Yaskawa INFORM job: DEMO_ROOF_UPPER_0625_3PAINT_22.JBI

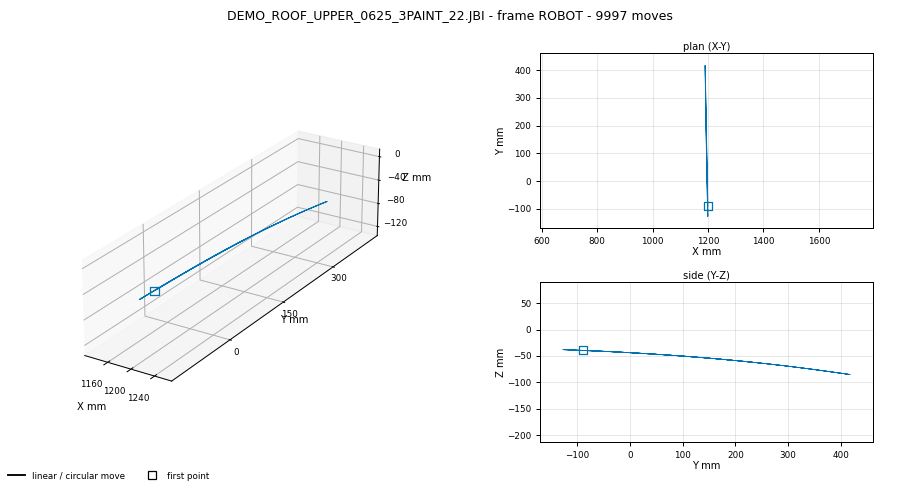
[picture p0: tool path of DEMO_ROOF_UPPER_0625_3PAINT_22.JBI in frame ROBOT, 9997 of 9997 moves have a stored position in this frame; points joined in program order, loops and branches not executed]
/JOB
//NAME DEMO_ROOF_UPPER_0625_3PAINT22
//POS
///NPOS 9997,0,0,0,0,0
///TOOL 0
///USER 0
///POSTYPE ROBOT
///RECTAN
///RCONF 1,0,0,0,0,0,0,0,0,0,0,0,0,0,0,0,0,0,0,0,0,0,0,0
C00000=1199.576,-89.571,-39.322,179.341,5.541,149.171
C00001=1199.572,-89.321,-39.332,179.344,5.541,149.171
C00002=1199.567,-89.072,-39.342,179.346,5.541,149.170
C00003=1199.562,-88.822,-39.354,179.348,5.541,149.169
C00004=1199.556,-88.573,-39.364,179.350,5.541,149.169
C00005=1199.551,-88.322,-39.375,179.353,5.541,149.168
C00006=1199.546,-88.073,-39.385,179.355,5.541,149.167
C00007=1199.540,-87.823,-39.395,179.357,5.542,149.167
C00008=1199.535,-87.573,-39.406,179.359,5.542,149.166
C00009=1199.530,-87.324,-39.416,179.362,5.542,149.165
C00010=1199.525,-87.074,-39.427,179.365,5.542,149.165
C00011=1199.519,-86.824,-39.437,179.366,5.542,149.164
C00012=1199.514,-86.574,-39.448,179.369,5.543,149.163
C00013=1199.509,-86.325,-39.458,179.371,5.542,149.163
C00014=1199.504,-86.075,-39.469,179.374,5.543,149.162
C00015=1199.498,-85.825,-39.480,179.375,5.543,149.162
C00016=1199.493,-85.575,-39.490,179.378,5.543,149.161
C00017=1199.488,-85.326,-39.500,179.381,5.544,149.160
C00018=1199.483,-85.076,-39.512,179.383,5.543,149.159
C00019=1199.477,-84.826,-39.522,179.385,5.544,149.159
C00020=1199.472,-84.576,-39.532,179.387,5.544,149.158
C00021=1199.467,-84.327,-39.543,179.390,5.544,149.158
C00022=1199.462,-84.077,-39.554,179.392,5.544,149.157
C00023=1199.457,-83.827,-39.564,179.394,5.545,149.156
C00024=1199.452,-83.577,-39.575,179.397,5.545,149.156
C00025=1199.446,-83.328,-39.586,179.399,5.545,149.155
C00026=1199.441,-83.078,-39.596,179.401,5.545,149.154
C00027=1199.436,-82.828,-39.606,179.403,5.545,149.154
C00028=1199.431,-82.579,-39.618,179.406,5.545,149.153
C00029=1199.425,-82.329,-39.628,179.408,5.545,149.152
C00030=1199.420,-82.079,-39.638,179.410,5.546,149.152
C00031=1199.415,-81.830,-39.649,179.412,5.546,149.151
C00032=1199.410,-81.580,-39.660,179.415,5.546,149.150
C00033=1199.404,-81.330,-39.670,179.417,5.546,149.150
C00034=1199.400,-81.081,-39.681,179.419,5.546,149.149
C00035=1199.394,-80.831,-39.692,179.422,5.547,149.149
C00036=1199.388,-80.581,-39.703,179.424,5.546,149.148
C00037=1199.383,-80.332,-39.714,179.426,5.547,149.147
C00038=1199.378,-80.081,-39.724,179.429,5.547,149.146
C00039=1199.373,-79.833,-39.735,179.431,5.547,149.146
C00040=1199.368,-79.582,-39.746,179.433,5.548,149.145
C00041=1199.362,-79.333,-39.756,179.435,5.547,149.145
C00042=1199.358,-79.083,-39.767,179.438,5.548,149.144
C00043=1199.353,-78.833,-39.778,179.440,5.548,149.143
C00044=1199.347,-78.584,-39.789,179.442,5.548,149.143
C00045=1199.342,-78.333,-39.800,179.445,5.549,149.142
C00046=1199.336,-78.084,-39.811,179.447,5.548,149.141
C00047=1199.331,-77.834,-39.821,179.450,5.549,149.140
C00048=1199.326,-77.585,-39.832,179.451,5.549,149.140
C00049=1199.321,-77.335,-39.843,179.454,5.549,149.139
C00050=1199.316,-77.085,-39.854,179.457,5.550,149.139
C00051=1199.310,-76.836,-39.865,179.459,5.549,149.138
C00052=1199.305,-76.585,-39.876,179.461,5.550,149.137
C00053=1199.300,-76.336,-39.887,179.463,5.550,149.137
C00054=1199.295,-76.086,-39.897,179.466,5.550,149.136
C00055=1199.289,-75.837,-39.908,179.468,5.550,149.135
C00056=1199.284,-75.566,-39.920,179.470,5.550,149.135
C00057=1199.278,-75.295,-39.933,179.473,5.551,149.134
C00058=1199.272,-75.024,-39.944,179.476,5.551,149.133
C00059=1199.267,-74.754,-39.955,179.478,5.551,149.132
C00060=1199.262,-74.504,-39.967,179.480,5.551,149.132
C00061=1199.256,-74.254,-39.977,179.483,5.552,149.131
C00062=1199.251,-74.005,-39.989,179.485,5.551,149.131
C00063=1199.246,-73.754,-39.999,179.487,5.552,149.130
C00064=1199.241,-73.505,-40.010,179.489,5.552,149.129
C00065=1199.235,-73.255,-40.022,179.492,5.552,149.129
C00066=1199.230,-73.006,-40.032,179.494,5.553,149.128
C00067=1199.225,-72.756,-40.044,179.496,5.552,149.127
C00068=1199.220,-72.506,-40.054,179.499,5.553,149.127
C00069=1199.214,-72.257,-40.066,179.501,5.554,149.126
C00070=1199.209,-72.007,-40.077,179.503,5.553,149.125
C00071=1199.204,-71.757,-40.088,179.506,5.554,149.125
C00072=1199.198,-71.508,-40.099,179.508,5.553,149.124
C00073=1199.194,-71.258,-40.110,179.511,5.554,149.123
C00074=1199.189,-71.008,-40.121,179.513,5.555,149.123
C00075=1199.183,-70.759,-40.132,179.515,5.554,149.122
C00076=1199.178,-70.508,-40.143,179.518,5.555,149.121
C00077=1199.173,-70.259,-40.154,179.520,5.554,149.121
C00078=1199.168,-70.010,-40.165,179.522,5.555,149.120
C00079=1199.162,-69.759,-40.176,179.525,5.556,149.119
C00080=1199.157,-69.510,-40.188,179.527,5.555,149.119
C00081=1199.152,-69.261,-40.199,179.529,5.556,149.118
C00082=1199.146,-69.011,-40.211,179.532,5.555,149.117
C00083=1199.141,-68.761,-40.221,179.534,5.556,149.117
C00084=1199.136,-68.512,-40.232,179.536,5.556,149.116
C00085=1199.131,-68.262,-40.244,179.538,5.556,149.115
C00086=1199.126,-68.011,-40.255,179.541,5.557,149.115
C00087=1199.121,-67.762,-40.266,179.544,5.557,149.114
C00088=1199.115,-67.513,-40.277,179.545,5.557,149.114
C00089=1199.110,-67.263,-40.289,179.548,5.557,149.113
C00090=1199.105,-67.013,-40.299,179.550,5.557,149.112
C00091=1199.099,-66.763,-40.311,179.553,5.557,149.111
C00092=1199.095,-66.514,-40.322,179.555,5.558,149.111
C00093=1199.089,-66.264,-40.334,179.557,5.558,149.110
C00094=1199.084,-66.014,-40.345,179.560,5.558,149.110
C00095=1199.079,-65.765,-40.355,179.562,5.559,149.109
C00096=1199.073,-65.515,-40.367,179.564,5.558,149.108
C00097=1199.069,-65.265,-40.379,179.567,5.559,149.108
C00098=1199.063,-65.015,-40.390,179.569,5.559,149.107
C00099=1199.058,-64.766,-40.401,179.571,5.559,149.106
C00100=1199.053,-64.516,-40.412,179.574,5.560,149.105
C00101=1199.048,-64.266,-40.424,179.576,5.559,149.105
C00102=1199.043,-64.017,-40.435,179.578,5.560,149.104
C00103=1199.037,-63.767,-40.447,179.581,5.561,149.104
C00104=1199.032,-63.518,-40.458,179.583,5.560,149.103
C00105=1199.027,-63.268,-40.470,179.586,5.561,149.102
C00106=1199.022,-63.018,-40.481,179.588,5.560,149.101
C00107=1199.016,-62.769,-40.491,179.590,5.561,149.101
C00108=1199.011,-62.519,-40.503,179.593,5.562,149.100
C00109=1199.006,-62.269,-40.515,179.595,5.561,149.100
C00110=1199.001,-62.019,-40.526,179.597,5.562,149.099
C00111=1198.996,-61.769,-40.538,179.600,5.562,149.098
C00112=1198.990,-61.520,-40.549,179.602,5.562,149.098
C00113=1198.985,-61.271,-40.560,179.604,5.563,149.097
C00114=1198.980,-61.021,-40.572,179.607,5.563,149.096
C00115=1198.975,-60.771,-40.584,179.609,5.563,149.096
C00116=1198.970,-60.521,-40.596,179.612,5.563,149.095
C00117=1198.965,-60.272,-40.606,179.614,5.564,149.094
C00118=1198.959,-60.022,-40.618,179.616,5.564,149.094
C00119=1198.955,-59.773,-40.630,179.619,5.564,149.093
C00120=1198.949,-59.523,-40.642,179.621,5.564,149.092
C00121=1198.944,-59.272,-40.652,179.623,5.564,149.092
C00122=1198.939,-59.022,-40.664,179.626,5.565,149.091
C00123=1198.933,-58.774,-40.675,179.628,5.565,149.090
C00124=1198.928,-58.524,-40.687,179.630,5.565,149.090
C00125=1198.923,-58.274,-40.698,179.633,5.565,149.089
C00126=1198.918,-58.025,-40.711,179.635,5.565,149.088
C00127=1198.913,-57.775,-40.723,179.637,5.566,149.088
C00128=1198.908,-57.525,-40.734,179.640,5.566,149.087
C00129=1198.902,-57.276,-40.745,179.642,5.566,149.086
C00130=1198.897,-57.026,-40.757,179.645,5.566,149.086
C00131=1198.892,-56.776,-40.769,179.647,5.567,149.085
C00132=1198.887,-56.527,-40.780,179.649,5.567,149.085
C00133=1198.882,-56.277,-40.792,179.652,5.567,149.084
C00134=1198.876,-56.027,-40.804,179.654,5.568,149.083
C00135=1198.872,-55.777,-40.815,179.656,5.567,149.082
C00136=1198.866,-55.527,-40.827,179.659,5.568,149.082
C00137=1198.861,-55.278,-40.838,179.661,5.569,149.081
C00138=1198.855,-55.028,-40.850,179.663,5.568,149.081
C00139=1198.850,-54.778,-40.861,179.666,5.569,149.080
C00140=1198.846,-54.529,-40.873,179.669,5.569,149.079
C00141=1198.840,-54.280,-40.885,179.671,5.569,149.078
C00142=1198.836,-54.030,-40.897,179.673,5.569,149.078
C00143=1198.830,-53.780,-40.909,179.676,5.570,149.077
C00144=1198.825,-53.530,-40.920,179.678,5.570,149.077
C00145=1198.820,-53.280,-40.932,179.680,5.570,149.076
C00146=1198.815,-53.030,-40.944,179.683,5.571,149.075
C00147=1198.809,-52.781,-40.956,179.685,5.570,149.074
C00148=1198.805,-52.531,-40.968,179.687,5.571,149.074
C00149=1198.799,-52.282,-40.979,179.690,5.572,149.073
C00150=1198.793,-52.032,-40.991,179.692,5.571,149.073
C00151=1198.789,-51.783,-41.002,179.695,5.572,149.072
C00152=1198.783,-51.533,-41.015,179.697,5.572,149.071
C00153=1198.778,-51.283,-41.027,179.699,5.572,149.071
C00154=1198.773,-51.034,-41.038,179.702,5.573,149.070
C00155=1198.768,-50.784,-41.050,179.704,5.573,149.069
C00156=1198.762,-50.534,-41.062,179.706,5.573,149.069
C00157=1198.757,-50.285,-41.074,179.709,5.573,149.068
C00158=1198.753,-50.035,-41.086,179.711,5.574,149.067
C00159=1198.747,-49.785,-41.098,179.713,5.574,149.067
C00160=1198.742,-49.515,-41.110,179.716,5.574,149.066
C00161=1198.736,-49.245,-41.123,179.719,5.575,149.065
C00162=1198.731,-48.975,-41.136,179.721,5.575,149.065
C00163=1198.725,-48.705,-41.149,179.724,5.575,149.064
C00164=1198.720,-48.456,-41.161,179.726,5.575,149.063
C00165=1198.714,-48.206,-41.173,179.729,5.576,149.062
C00166=1198.709,-47.956,-41.185,179.731,5.576,149.062
C00167=1198.704,-47.706,-41.196,179.733,5.576,149.061
C00168=1198.699,-47.457,-41.209,179.736,5.576,149.060
C00169=1198.694,-47.207,-41.221,179.738,5.577,149.060
C00170=1198.688,-46.957,-41.233,179.741,5.577,149.059
C00171=1198.683,-46.708,-41.245,179.743,5.577,149.058
C00172=1198.678,-46.458,-41.257,179.746,5.577,149.058
C00173=1198.673,-46.209,-41.269,179.748,5.578,149.057
C00174=1198.668,-45.959,-41.281,179.750,5.578,149.057
C00175=1198.662,-45.709,-41.293,179.753,5.578,149.056
C00176=1198.657,-45.460,-41.306,179.755,5.579,149.055
C00177=1198.653,-45.210,-41.317,179.757,5.578,149.054
C00178=1198.647,-44.960,-41.329,179.760,5.579,149.054
C00179=1198.642,-44.711,-41.341,179.763,5.579,149.053
C00180=1198.637,-44.461,-41.353,179.764,5.579,149.053
C00181=1198.632,-44.211,-41.366,179.767,5.580,149.052
C00182=1198.627,-43.961,-41.378,179.770,5.580,149.051
C00183=1198.622,-43.712,-41.390,179.772,5.581,149.051
C00184=1198.617,-43.462,-41.402,179.774,5.580,149.050
C00185=1198.611,-43.212,-41.414,179.777,5.581,149.049
C00186=1198.606,-42.963,-41.426,179.779,5.582,149.049
C00187=1198.601,-42.713,-41.438,179.781,5.581,149.048
C00188=1198.596,-42.463,-41.451,179.784,5.582,149.047
C00189=1198.590,-42.213,-41.463,179.787,5.582,149.047
C00190=1198.585,-41.964,-41.475,179.789,5.583,149.046
C00191=1198.580,-41.714,-41.487,179.791,5.583,149.045
C00192=1198.575,-41.465,-41.499,179.794,5.583,149.045
C00193=1198.570,-41.215,-41.511,179.796,5.584,149.044
C00194=1198.565,-40.966,-41.524,179.798,5.583,149.043
C00195=1198.559,-40.716,-41.536,179.801,5.584,149.043
C00196=1198.555,-40.466,-41.549,179.804,5.584,149.042
C00197=1198.549,-40.216,-41.561,179.806,5.585,149.041
C00198=1198.544,-39.967,-41.573,179.808,5.585,149.041
C00199=1198.539,-39.717,-41.586,179.811,5.585,149.040
C00200=1198.534,-39.467,-41.598,179.813,5.586,149.039
C00201=1198.529,-39.218,-41.610,179.815,5.585,149.039
C00202=1198.523,-38.968,-41.622,179.817,5.586,149.038
C00203=1198.518,-38.719,-41.635,179.820,5.587,149.037
C00204=1198.513,-38.469,-41.647,179.823,5.587,149.037
C00205=1198.507,-38.220,-41.659,179.825,5.587,149.036
C00206=1198.503,-37.970,-41.672,179.828,5.587,149.035
C00207=1198.497,-37.720,-41.684,179.830,5.588,149.035
C00208=1198.492,-37.470,-41.697,179.832,5.588,149.034
C00209=1198.487,-37.221,-41.709,179.834,5.588,149.033
C00210=1198.482,-36.971,-41.721,179.837,5.589,149.033
C00211=1198.477,-36.722,-41.734,179.840,5.589,149.032
C00212=1198.471,-36.472,-41.746,179.842,5.589,149.031
C00213=1198.467,-36.222,-41.759,179.845,5.589,149.031
C00214=1198.462,-35.973,-41.771,179.847,5.590,149.030
C00215=1198.456,-35.723,-41.783,179.849,5.590,149.029
C00216=1198.451,-35.473,-41.796,179.851,5.590,149.029
C00217=1198.446,-35.224,-41.808,179.854,5.591,149.028
C00218=1198.441,-34.975,-41.821,179.857,5.591,149.027
C00219=1198.436,-34.724,-41.833,179.859,5.592,149.027
C00220=1198.431,-34.475,-41.846,179.861,5.592,149.026
C00221=1198.426,-34.225,-41.858,179.864,5.592,149.026
C00222=1198.420,-33.975,-41.870,179.866,5.592,149.025
C00223=1198.415,-33.726,-41.883,179.869,5.593,149.024
C00224=1198.410,-33.477,-41.895,179.871,5.593,149.023
C00225=1198.406,-33.227,-41.908,179.873,5.593,149.023
C00226=1198.400,-32.977,-41.920,179.876,5.594,149.022
C00227=1198.395,-32.728,-41.933,179.879,5.594,149.022
C00228=1198.389,-32.478,-41.946,179.881,5.594,149.021
C00229=1198.384,-32.229,-41.959,179.883,5.594,149.020
C00230=1198.379,-31.978,-41.971,179.886,5.595,149.019
C00231=1198.374,-31.729,-41.984,179.888,5.596,149.019
C00232=1198.369,-31.479,-41.996,179.890,5.595,149.018
C00233=1198.364,-31.230,-42.009,179.893,5.596,149.018
C00234=1198.359,-30.980,-42.022,179.896,5.596,149.017
C00235=1198.354,-30.731,-42.034,179.898,5.597,149.016
C00236=1198.349,-30.481,-42.046,179.900,5.597,149.016
C00237=1198.343,-30.231,-42.059,179.902,5.597,149.015
C00238=1198.338,-29.982,-42.072,179.905,5.598,149.014
C00239=1198.333,-29.732,-42.085,179.908,5.598,149.014
C00240=1198.328,-29.482,-42.098,179.910,5.598,149.013
C00241=1198.323,-29.233,-42.110,179.913,5.598,149.012
C00242=1198.318,-28.984,-42.123,179.915,5.599,149.012
C00243=1198.312,-28.733,-42.136,179.917,5.600,149.011
C00244=1198.307,-28.484,-42.148,179.919,5.599,149.010
C00245=1198.302,-28.234,-42.161,179.922,5.600,149.010
C00246=1198.298,-27.984,-42.174,179.925,5.600,149.009
C00247=1198.292,-27.735,-42.186,179.927,5.601,149.008
C00248=1198.287,-27.485,-42.200,179.929,5.601,149.008
C00249=1198.281,-27.236,-42.212,179.932,5.601,149.007
C00250=1198.277,-26.986,-42.225,179.934,5.602,149.006
C00251=1198.272,-26.737,-42.238,179.937,5.602,149.006
C00252=1198.267,-26.487,-42.250,179.940,5.603,149.005
C00253=1198.261,-26.237,-42.264,179.942,5.602,149.004
C00254=1198.256,-25.988,-42.276,179.944,5.603,149.004
C00255=1198.251,-25.738,-42.289,179.947,5.604,149.003
C00256=1198.246,-25.489,-42.302,179.949,5.604,149.002
C00257=1198.241,-25.239,-42.315,179.951,5.604,149.002
C00258=1198.236,-24.989,-42.328,179.954,5.604,149.001
C00259=1198.230,-24.740,-42.340,179.956,5.605,149.001
C00260=1198.226,-24.490,-42.353,179.959,5.606,149.000
C00261=1198.220,-24.240,-42.367,179.961,5.606,148.999
C00262=1198.215,-23.991,-42.379,179.964,5.606,148.999
C00263=1198.210,-23.741,-42.392,179.966,5.606,148.998
C00264=1198.204,-23.472,-42.406,179.969,5.607,148.997
C00265=1198.199,-23.202,-42.420,179.972,5.607,148.996
C00266=1198.193,-22.932,-42.434,179.974,5.608,148.996
C00267=1198.188,-22.662,-42.448,179.977,5.608,148.995
C00268=1198.183,-22.413,-42.462,179.980,5.608,148.994
C00269=1198.178,-22.164,-42.474,179.982,5.608,148.994
C00270=1198.173,-21.914,-42.487,179.984,5.609,148.993
C00271=1198.167,-21.664,-42.500,179.986,5.609,148.992
C00272=1198.162,-21.415,-42.513,179.989,5.610,148.992
C00273=1198.158,-21.165,-42.526,179.992,5.610,148.991
C00274=1198.152,-20.915,-42.539,179.994,5.610,148.990
C00275=1198.147,-20.666,-42.552,179.996,5.611,148.990
C00276=1198.142,-20.416,-42.565,179.999,5.611,148.989
C00277=1198.137,-20.167,-42.579,-179.999,5.612,148.989
C00278=1198.132,-19.917,-42.592,-179.996,5.612,148.988
C00279=1198.127,-19.668,-42.604,-179.994,5.612,148.987
C00280=1198.121,-19.418,-42.617,-179.991,5.612,148.986
C00281=1198.117,-19.168,-42.630,-179.989,5.613,148.986
C00282=1198.111,-18.918,-42.644,-179.986,5.614,148.985
C00283=1198.106,-18.670,-42.657,-179.984,5.614,148.985
C00284=1198.101,-18.420,-42.670,-179.982,5.614,148.984
C00285=1198.095,-18.170,-42.683,-179.979,5.614,148.983
C00286=1198.091,-17.920,-42.696,-179.976,5.615,148.983
C00287=1198.085,-17.671,-42.710,-179.974,5.615,148.982
C00288=1198.081,-17.421,-42.723,-179.972,5.616,148.981
C00289=1198.076,-17.172,-42.735,-179.970,5.616,148.981
C00290=1198.070,-16.922,-42.749,-179.967,5.616,148.980
C00291=1198.066,-16.673,-42.762,-179.964,5.617,148.979
C00292=1198.060,-16.423,-42.776,-179.962,5.617,148.979
C00293=1198.055,-16.173,-42.789,-179.959,5.618,148.978
C00294=1198.049,-15.923,-42.802,-179.957,5.619,148.977
C00295=1198.045,-15.674,-42.815,-179.955,5.618,148.977
C00296=1198.039,-15.424,-42.829,-179.952,5.619,148.976
C00297=1198.035,-15.174,-42.842,-179.949,5.619,148.975
C00298=1198.029,-14.925,-42.855,-179.947,5.620,148.975
C00299=1198.024,-14.676,-42.868,-179.944,5.621,148.974
C00300=1198.019,-14.426,-42.882,-179.942,5.620,148.973
C00301=1198.014,-14.177,-42.895,-179.940,5.621,148.973
C00302=1198.009,-13.927,-42.909,-179.937,5.621,148.972
C00303=1198.004,-13.677,-42.921,-179.934,5.622,148.971
C00304=1197.999,-13.428,-42.935,-179.932,5.623,148.971
C00305=1197.994,-13.178,-42.948,-179.930,5.623,148.970
C00306=1197.988,-12.928,-42.962,-179.928,5.623,148.970
C00307=1197.984,-12.679,-42.975,-179.925,5.623,148.969
C00308=1197.978,-12.429,-42.988,-179.922,5.624,148.968
C00309=1197.973,-12.180,-43.002,-179.920,5.624,148.967
C00310=1197.968,-11.930,-43.015,-179.917,5.625,148.967
C00311=1197.963,-11.681,-43.028,-179.915,5.625,148.966
C00312=1197.958,-11.431,-43.042,-179.913,5.625,148.966
C00313=1197.953,-11.181,-43.055,-179.910,5.626,148.965
C00314=1197.948,-10.932,-43.069,-179.907,5.626,148.964
C00315=1197.942,-10.682,-43.082,-179.905,5.627,148.964
C00316=1197.938,-10.433,-43.096,-179.903,5.627,148.963
C00317=1197.932,-10.183,-43.109,-179.900,5.628,148.962
C00318=1197.928,-9.934,-43.123,-179.897,5.628,148.962
C00319=1197.923,-9.683,-43.136,-179.895,5.628,148.961
C00320=1197.917,-9.434,-43.150,-179.892,5.629,148.960
C00321=1197.913,-9.184,-43.163,-179.890,5.629,148.960
C00322=1197.907,-8.935,-43.177,-179.888,5.630,148.959
C00323=1197.902,-8.685,-43.190,-179.885,5.630,148.958
C00324=1197.897,-8.436,-43.204,-179.882,5.631,148.958
C00325=1197.892,-8.186,-43.218,-179.880,5.631,148.957
C00326=1197.887,-7.937,-43.231,-179.878,5.631,148.956
C00327=1197.882,-7.687,-43.244,-179.875,5.632,148.956
C00328=1197.877,-7.438,-43.258,-179.873,5.632,148.955
C00329=1197.872,-7.188,-43.271,-179.870,5.633,148.955
C00330=1197.867,-6.938,-43.286,-179.867,5.633,148.954
C00331=1197.861,-6.689,-43.298,-179.865,5.634,148.953
C00332=1197.856,-6.439,-43.313,-179.863,5.634,148.953
C00333=1197.852,-6.189,-43.327,-179.861,5.634,148.952
C00334=1197.846,-5.940,-43.339,-179.858,5.635,148.951
C00335=1197.841,-5.690,-43.354,-179.855,5.635,148.951
C00336=1197.836,-5.441,-43.367,-179.853,5.636,148.950
C00337=1197.831,-5.191,-43.381,-179.850,5.636,148.949
C00338=1197.826,-4.942,-43.395,-179.848,5.637,148.949
C00339=1197.821,-4.692,-43.408,-179.846,5.637,148.948
C00340=1197.816,-4.442,-43.422,-179.843,5.637,148.947
C00341=1197.811,-4.194,-43.436,-179.840,5.638,148.947
C00342=1197.806,-3.943,-43.449,-179.838,5.638,148.946
C00343=1197.801,-3.694,-43.463,-179.836,5.639,148.946
C00344=1197.795,-3.445,-43.477,-179.833,5.640,148.945
C00345=1197.790,-3.195,-43.490,-179.830,5.640,148.944
C00346=1197.786,-2.945,-43.505,-179.828,5.641,148.944
C00347=1197.780,-2.696,-43.519,-179.826,5.640,148.943
C00348=1197.775,-2.446,-43.532,-179.823,5.641,148.942
C00349=1197.770,-2.197,-43.545,-179.821,5.642,148.942
C00350=1197.765,-1.947,-43.560,-179.818,5.642,148.941
C00351=1197.760,-1.697,-43.574,-179.815,5.643,148.940
C00352=1197.754,-1.448,-43.587,-179.813,5.643,148.940
C00353=1197.750,-1.198,-43.601,-179.810,5.644,148.939
C00354=1197.745,-0.949,-43.615,-179.808,5.644,148.938
C00355=1197.739,-0.700,-43.629,-179.806,5.644,148.938
C00356=1197.734,-0.449,-43.643,-179.803,5.645,148.937
C00357=1197.729,-0.200,-43.657,-179.801,5.645,148.936
C00358=1197.724,0.050,-43.671,-179.798,5.646,148.936
C00359=1197.719,0.299,-43.684,-179.796,5.646,148.935
C00360=1197.714,0.548,-43.699,-179.793,5.647,148.935
C00361=1197.709,0.799,-43.712,-179.790,5.647,148.934
C00362=1197.704,1.048,-43.726,-179.788,5.648,148.933
C00363=1197.699,1.298,-43.740,-179.785,5.648,148.932
C00364=1197.694,1.547,-43.755,-179.783,5.649,148.932
C00365=1197.689,1.796,-43.768,-179.781,5.649,148.931
C00366=1197.684,2.046,-43.782,-179.778,5.649,148.931
C00367=1197.679,2.296,-43.796,-179.776,5.650,148.930
C00368=1197.674,2.565,-43.812,-179.773,5.650,148.929
C00369=1197.668,2.833,-43.826,-179.770,5.651,148.929
C00370=1197.662,3.103,-43.841,-179.768,5.651,148.928
C00371=1197.657,3.372,-43.857,-179.765,5.652,148.927
C00372=1197.652,3.622,-43.871,-179.762,5.652,148.927
C00373=1197.647,3.872,-43.885,-179.760,5.653,148.926
C00374=1197.641,4.121,-43.899,-179.758,5.654,148.925
C00375=1197.636,4.370,-43.913,-179.755,5.654,148.925
C00376=1197.631,4.620,-43.927,-179.752,5.655,148.924
C00377=1197.626,4.870,-43.942,-179.750,5.655,148.923
C00378=1197.621,5.119,-43.955,-179.747,5.656,148.923
C00379=1197.617,5.368,-43.969,-179.745,5.657,148.922
C00380=1197.612,5.618,-43.983,-179.742,5.657,148.921
C00381=1197.607,5.868,-43.998,-179.739,5.658,148.921
C00382=1197.601,6.117,-44.012,-179.737,5.657,148.920
C00383=1197.596,6.366,-44.026,-179.735,5.658,148.919
C00384=1197.591,6.616,-44.040,-179.733,5.659,148.919
C00385=1197.586,6.866,-44.054,-179.730,5.659,148.918
C00386=1197.581,7.116,-44.069,-179.727,5.660,148.918
C00387=1197.576,7.365,-44.083,-179.725,5.660,148.917
C00388=1197.571,7.614,-44.097,-179.722,5.661,148.916
C00389=1197.566,7.864,-44.111,-179.720,5.661,148.916
C00390=1197.561,8.114,-44.125,-179.717,5.662,148.915
C00391=1197.556,8.363,-44.140,-179.714,5.662,148.914
C00392=1197.550,8.612,-44.154,-179.712,5.663,148.914
C00393=1197.545,8.862,-44.168,-179.709,5.663,148.913
C00394=1197.540,9.112,-44.182,-179.707,5.664,148.913
C00395=1197.536,9.361,-44.197,-179.705,5.664,148.912
C00396=1197.531,9.611,-44.211,-179.702,5.664,148.911
C00397=1197.526,9.860,-44.226,-179.700,5.665,148.911
C00398=1197.520,10.109,-44.240,-179.697,5.665,148.910
C00399=1197.515,10.359,-44.254,-179.695,5.666,148.909
C00400=1197.510,10.609,-44.268,-179.692,5.667,148.909
C00401=1197.505,10.859,-44.283,-179.690,5.667,148.908
C00402=1197.500,11.108,-44.297,-179.687,5.668,148.907
C00403=1197.495,11.358,-44.312,-179.685,5.669,148.907
C00404=1197.490,11.607,-44.326,-179.682,5.669,148.906
C00405=1197.485,11.856,-44.341,-179.679,5.670,148.905
C00406=1197.480,12.106,-44.355,-179.677,5.670,148.905
C00407=1197.475,12.356,-44.369,-179.674,5.671,148.904
C00408=1197.470,12.605,-44.383,-179.672,5.672,148.904
C00409=1197.465,12.855,-44.398,-179.669,5.672,148.903
C00410=1197.460,13.104,-44.413,-179.667,5.673,148.902
C00411=1197.454,13.354,-44.427,-179.664,5.673,148.902
C00412=1197.449,13.603,-44.441,-179.662,5.673,148.901
C00413=1197.444,13.852,-44.456,-179.660,5.674,148.900
C00414=1197.439,14.102,-44.471,-179.657,5.674,148.900
C00415=1197.434,14.352,-44.485,-179.654,5.675,148.899
C00416=1197.429,14.601,-44.499,-179.652,5.675,148.898
C00417=1197.425,14.851,-44.514,-179.649,5.676,148.898
C00418=1197.419,15.101,-44.529,-179.647,5.676,148.897
C00419=1197.414,15.350,-44.543,-179.644,5.677,148.897
C00420=1197.409,15.599,-44.558,-179.642,5.677,148.896
C00421=1197.404,15.849,-44.573,-179.639,5.678,148.895
C00422=1197.400,16.099,-44.587,-179.637,5.679,148.895
C00423=1197.394,16.348,-44.601,-179.634,5.679,148.894
C00424=1197.389,16.597,-44.616,-179.632,5.680,148.893
C00425=1197.384,16.847,-44.631,-179.629,5.680,148.893
C00426=1197.379,17.097,-44.645,-179.626,5.681,148.892
C00427=1197.374,17.346,-44.660,-179.624,5.682,148.892
C00428=1197.369,17.595,-44.674,-179.622,5.682,148.891
C00429=1197.364,17.845,-44.690,-179.619,5.683,148.890
C00430=1197.359,18.095,-44.704,-179.616,5.683,148.890
C00431=1197.354,18.344,-44.718,-179.614,5.684,148.889
C00432=1197.349,18.593,-44.733,-179.611,5.685,148.888
C00433=1197.343,18.843,-44.748,-179.609,5.685,148.888
C00434=1197.339,19.092,-44.763,-179.606,5.686,148.887
C00435=1197.334,19.342,-44.778,-179.603,5.686,148.886
C00436=1197.329,19.592,-44.792,-179.601,5.687,148.886
C00437=1197.323,19.841,-44.807,-179.599,5.688,148.885
C00438=1197.319,20.091,-44.822,-179.596,5.688,148.885
C00439=1197.314,20.340,-44.837,-179.593,5.689,148.884
C00440=1197.308,20.590,-44.852,-179.591,5.689,148.883
C00441=1197.304,20.839,-44.867,-179.589,5.690,148.883
C00442=1197.299,21.089,-44.881,-179.586,5.690,148.882
C00443=1197.294,21.338,-44.896,-179.583,5.691,148.881
C00444=1197.288,21.588,-44.911,-179.581,5.691,148.881
C00445=1197.284,21.837,-44.926,-179.578,5.692,148.880
C00446=1197.279,22.087,-44.940,-179.576,5.693,148.880
C00447=1197.273,22.336,-44.956,-179.573,5.693,148.879
C00448=1197.268,22.586,-44.970,-179.571,5.694,148.878
C00449=1197.264,22.835,-44.985,-179.568,5.695,148.878
C00450=1197.258,23.085,-45.000,-179.566,5.695,148.877
C00451=1197.253,23.334,-45.015,-179.563,5.696,148.876
C00452=1197.248,23.584,-45.030,-179.560,5.696,148.876
C00453=1197.243,23.833,-45.045,-179.558,5.697,148.875
C00454=1197.238,24.082,-45.060,-179.556,5.698,148.875
C00455=1197.233,24.332,-45.074,-179.553,5.698,148.874
C00456=1197.228,24.581,-45.089,-179.550,5.699,148.873
C00457=1197.223,24.831,-45.104,-179.548,5.699,148.873
C00458=1197.218,25.081,-45.120,-179.546,5.700,148.872
C00459=1197.214,25.330,-45.135,-179.543,5.701,148.871
C00460=1197.208,25.580,-45.149,-179.540,5.701,148.871
C00461=1197.203,25.830,-45.164,-179.538,5.702,148.870
C00462=1197.199,26.079,-45.179,-179.535,5.702,148.870
C00463=1197.193,26.329,-45.194,-179.533,5.703,148.869
C00464=1197.188,26.578,-45.209,-179.530,5.703,148.868
C00465=1197.183,26.827,-45.225,-179.527,5.704,148.868
C00466=1197.178,27.077,-45.239,-179.525,5.705,148.867
C00467=1197.173,27.326,-45.255,-179.523,5.705,148.866
C00468=1197.168,27.575,-45.270,-179.520,5.706,148.866
C00469=1197.163,27.826,-45.285,-179.517,5.706,148.865
C00470=1197.158,28.075,-45.300,-179.515,5.707,148.865
C00471=1197.153,28.325,-45.316,-179.513,5.708,148.864
C00472=1197.148,28.593,-45.331,-179.510,5.708,148.863
C00473=1197.142,28.862,-45.348,-179.507,5.709,148.863
C00474=1197.137,29.131,-45.364,-179.505,5.709,148.862
C00475=1197.131,29.400,-45.380,-179.501,5.711,148.861
C00476=1197.126,29.649,-45.395,-179.499,5.711,148.861
C00477=1197.121,29.898,-45.411,-179.496,5.712,148.860
C00478=1197.116,30.147,-45.426,-179.494,5.713,148.859
C00479=1197.111,30.397,-45.441,-179.491,5.713,148.859
C00480=1197.107,30.647,-45.456,-179.489,5.714,148.858
C00481=1197.101,30.896,-45.472,-179.486,5.714,148.857
C00482=1197.097,31.146,-45.487,-179.484,5.715,148.857
C00483=1197.091,31.395,-45.502,-179.481,5.715,148.856
C00484=1197.086,31.644,-45.518,-179.479,5.716,148.856
C00485=1197.081,31.894,-45.532,-179.476,5.717,148.855
C00486=1197.076,32.144,-45.548,-179.474,5.717,148.854
C00487=1197.071,32.393,-45.563,-179.471,5.718,148.854
C00488=1197.066,32.643,-45.579,-179.469,5.718,148.853
C00489=1197.061,32.892,-45.594,-179.466,5.719,148.852
C00490=1197.056,33.141,-45.609,-179.464,5.720,148.852
C00491=1197.051,33.391,-45.625,-179.461,5.720,148.851
C00492=1197.047,33.640,-45.640,-179.458,5.721,148.851
C00493=1197.041,33.890,-45.655,-179.456,5.721,148.850
C00494=1197.036,34.139,-45.670,-179.454,5.722,148.850
C00495=1197.031,34.389,-45.686,-179.450,5.724,148.849
C00496=1197.026,34.639,-45.702,-179.448,5.724,148.848
C00497=1197.021,34.888,-45.717,-179.445,5.725,148.847
C00498=1197.016,35.138,-45.732,-179.443,5.726,148.847
C00499=1197.011,35.387,-45.748,-179.440,5.726,148.846
C00500=1197.007,35.637,-45.763,-179.438,5.727,148.846
C00501=1197.001,35.886,-45.779,-179.435,5.727,148.845
C00502=1196.997,36.135,-45.794,-179.433,5.728,148.845
C00503=1196.991,36.385,-45.809,-179.430,5.728,148.844
C00504=1196.986,36.635,-45.825,-179.428,5.729,148.843
C00505=1196.981,36.884,-45.841,-179.425,5.730,148.843
C00506=1196.976,37.133,-45.856,-179.423,5.730,148.842
C00507=1196.971,37.383,-45.871,-179.420,5.731,148.841
C00508=1196.966,37.633,-45.887,-179.418,5.731,148.841
C00509=1196.962,37.882,-45.902,-179.415,5.732,148.840
C00510=1196.956,38.131,-45.918,-179.412,5.734,148.840
C00511=1196.951,38.381,-45.934,-179.409,5.734,148.839
C00512=1196.947,38.630,-45.949,-179.407,5.735,148.838
C00513=1196.942,38.879,-45.965,-179.405,5.736,148.838
C00514=1196.936,39.129,-45.981,-179.402,5.736,148.837
C00515=1196.931,39.378,-45.996,-179.399,5.737,148.836
C00516=1196.927,39.628,-46.012,-179.397,5.738,148.836
C00517=1196.921,39.877,-46.027,-179.395,5.738,148.835
C00518=1196.916,40.127,-46.043,-179.392,5.739,148.835
C00519=1196.911,40.377,-46.059,-179.389,5.739,148.834
C00520=1196.907,40.626,-46.074,-179.387,5.740,148.834
C00521=1196.901,40.875,-46.089,-179.385,5.741,148.833
C00522=1196.897,41.125,-46.106,-179.381,5.742,148.832
C00523=1196.891,41.374,-46.122,-179.379,5.742,148.832
C00524=1196.886,41.623,-46.137,-179.377,5.743,148.831
C00525=1196.882,41.873,-46.153,-179.374,5.744,148.830
C00526=1196.877,42.123,-46.168,-179.371,5.744,148.830
C00527=1196.871,42.371,-46.185,-179.369,5.745,148.829
C00528=1196.867,42.622,-46.201,-179.366,5.746,148.829
C00529=1196.861,42.871,-46.216,-179.364,5.746,148.828
C00530=1196.856,43.120,-46.232,-179.361,5.747,148.827
C00531=1196.852,43.370,-46.248,-179.359,5.748,148.827
C00532=1196.847,43.619,-46.263,-179.356,5.749,148.826
C00533=1196.841,43.868,-46.279,-179.353,5.750,148.826
C00534=1196.837,44.118,-46.295,-179.351,5.750,148.825
C00535=1196.831,44.367,-46.311,-179.348,5.751,148.824
C00536=1196.826,44.617,-46.327,-179.346,5.751,148.824
C00537=1196.821,44.867,-46.343,-179.343,5.752,148.823
C00538=1196.817,45.116,-46.358,-179.341,5.753,148.823
C00539=1196.812,45.365,-46.374,-179.338,5.753,148.822
C00540=1196.807,45.615,-46.390,-179.336,5.754,148.821
C00541=1196.801,45.864,-46.406,-179.333,5.756,148.821
C00542=1196.797,46.114,-46.422,-179.330,5.756,148.820
C00543=1196.792,46.363,-46.438,-179.328,5.757,148.820
C00544=1196.787,46.613,-46.454,-179.325,5.757,148.819
C00545=1196.782,46.862,-46.470,-179.323,5.758,148.818
C00546=1196.776,47.111,-46.486,-179.320,5.759,148.818
C00547=1196.772,47.361,-46.502,-179.318,5.759,148.817
C00548=1196.766,47.610,-46.518,-179.315,5.760,148.817
C00549=1196.762,47.860,-46.533,-179.312,5.761,148.816
C00550=1196.757,48.109,-46.550,-179.310,5.762,148.815
C00551=1196.753,48.359,-46.566,-179.307,5.763,148.815
C00552=1196.747,48.608,-46.582,-179.305,5.763,148.814
C00553=1196.742,48.857,-46.597,-179.302,5.764,148.813
C00554=1196.737,49.107,-46.613,-179.300,5.764,148.813
C00555=1196.732,49.356,-46.630,-179.297,5.765,148.812
C00556=1196.727,49.606,-46.646,-179.295,5.766,148.812
C00557=1196.722,49.855,-46.662,-179.292,5.767,148.811
C00558=1196.718,50.105,-46.678,-179.289,5.768,148.811
C00559=1196.712,50.354,-46.694,-179.287,5.769,148.810
C00560=1196.708,50.604,-46.710,-179.284,5.769,148.809
C00561=1196.703,50.853,-46.726,-179.282,5.770,148.809
C00562=1196.698,51.103,-46.742,-179.279,5.771,148.808
C00563=1196.693,51.351,-46.759,-179.277,5.771,148.807
C00564=1196.688,51.602,-46.775,-179.273,5.772,148.807
C00565=1196.683,51.850,-46.791,-179.271,5.773,148.806
C00566=1196.678,52.100,-46.807,-179.269,5.774,148.806
C00567=1196.673,52.349,-46.823,-179.266,5.774,148.805
C00568=1196.669,52.599,-46.840,-179.264,5.775,148.805
C00569=1196.662,52.848,-46.856,-179.261,5.776,148.804
C00570=1196.658,53.098,-46.873,-179.258,5.777,148.803
C00571=1196.653,53.347,-46.888,-179.256,5.778,148.803
C00572=1196.648,53.597,-46.905,-179.253,5.779,148.802
C00573=1196.643,53.846,-46.921,-179.251,5.779,148.802
C00574=1196.638,54.096,-46.937,-179.248,5.780,148.801
C00575=1196.633,54.344,-46.954,-179.246,5.781,148.800
C00576=1196.628,54.614,-46.971,-179.243,5.782,148.800
C00577=1196.623,54.881,-46.989,-179.240,5.782,148.799
C00578=1196.617,55.150,-47.006,-179.237,5.783,148.798
C00579=1196.612,55.419,-47.024,-179.234,5.784,148.798
C00580=1196.607,55.668,-47.040,-179.232,5.785,148.797
C00581=1196.602,55.918,-47.057,-179.229,5.786,148.797
C00582=1196.597,56.167,-47.073,-179.227,5.786,148.796
C00583=1196.592,56.417,-47.089,-179.225,5.787,148.796
C00584=1196.586,56.666,-47.106,-179.221,5.789,148.795
C00585=1196.582,56.915,-47.122,-179.219,5.789,148.794
C00586=1196.577,57.165,-47.138,-179.217,5.790,148.794
C00587=1196.572,57.414,-47.155,-179.214,5.791,148.793
C00588=1196.568,57.664,-47.171,-179.211,5.791,148.792
C00589=1196.562,57.913,-47.188,-179.209,5.792,148.792
C00590=1196.557,58.163,-47.204,-179.206,5.793,148.791
C00591=1196.552,58.412,-47.221,-179.203,5.794,148.791
C00592=1196.547,58.661,-47.237,-179.201,5.795,148.790
C00593=1196.543,58.911,-47.254,-179.199,5.795,148.790
C00594=1196.537,59.160,-47.271,-179.196,5.796,148.789
C00595=1196.532,59.410,-47.287,-179.193,5.798,148.788
C00596=1196.528,59.659,-47.303,-179.191,5.798,148.788
C00597=1196.523,59.908,-47.320,-179.188,5.799,148.787
C00598=1196.518,60.158,-47.337,-179.186,5.800,148.787
C00599=1196.512,60.407,-47.353,-179.183,5.800,148.786
C00600=1196.508,60.656,-47.370,-179.180,5.801,148.785
C00601=1196.503,60.906,-47.386,-179.178,5.802,148.785
C00602=1196.497,61.155,-47.403,-179.175,5.803,148.784
C00603=1196.493,61.405,-47.419,-179.172,5.803,148.784
C00604=1196.488,61.654,-47.436,-179.170,5.804,148.783
C00605=1196.483,61.903,-47.453,-179.167,5.806,148.783
C00606=1196.478,62.153,-47.470,-179.164,5.806,148.782
C00607=1196.474,62.402,-47.486,-179.162,5.807,148.781
C00608=1196.469,62.651,-47.503,-179.160,5.808,148.781
C00609=1196.463,62.901,-47.520,-179.158,5.809,148.780
C00610=1196.459,63.150,-47.537,-179.154,5.810,148.780
C00611=1196.454,63.399,-47.553,-179.152,5.810,148.779
C00612=1196.449,63.649,-47.570,-179.150,5.811,148.779
C00613=1196.444,63.899,-47.586,-179.147,5.812,148.778
C00614=1196.439,64.148,-47.602,-179.144,5.813,148.777
C00615=1196.433,64.398,-47.620,-179.142,5.814,148.777
C00616=1196.429,64.647,-47.636,-179.139,5.815,148.776
C00617=1196.424,64.896,-47.653,-179.136,5.815,148.775
C00618=1196.419,65.146,-47.670,-179.134,5.816,148.775
C00619=1196.414,65.395,-47.687,-179.131,5.817,148.774
C00620=1196.409,65.644,-47.705,-179.128,5.818,148.774
C00621=1196.404,65.893,-47.721,-179.126,5.819,148.773
C00622=1196.400,66.143,-47.738,-179.124,5.819,148.773
C00623=1196.395,66.392,-47.755,-179.121,5.821,148.772
C00624=1196.390,66.642,-47.772,-179.118,5.822,148.772
C00625=1196.384,66.891,-47.788,-179.116,5.822,148.771
C00626=1196.380,67.140,-47.805,-179.113,5.823,148.770
C00627=1196.375,67.390,-47.822,-179.111,5.824,148.770
C00628=1196.369,67.639,-47.839,-179.108,5.825,148.769
C00629=1196.365,67.889,-47.855,-179.105,5.826,148.769
C00630=1196.360,68.138,-47.873,-179.103,5.827,148.768
C00631=1196.355,68.388,-47.889,-179.100,5.827,148.767
C00632=1196.350,68.637,-47.907,-179.097,5.829,148.767
C00633=1196.345,68.886,-47.924,-179.095,5.829,148.766
C00634=1196.340,69.136,-47.941,-179.093,5.830,148.766
C00635=1196.336,69.385,-47.957,-179.090,5.831,148.765
C00636=1196.330,69.635,-47.975,-179.087,5.832,148.765
C00637=1196.325,69.884,-47.991,-179.085,5.833,148.764
C00638=1196.320,70.133,-48.009,-179.082,5.834,148.763
C00639=1196.316,70.382,-48.026,-179.080,5.835,148.763
C00640=1196.311,70.632,-48.043,-179.077,5.836,148.762
C00641=1196.306,70.882,-48.060,-179.074,5.836,148.762
C00642=1196.301,71.130,-48.077,-179.072,5.837,148.761
C00643=1196.296,71.379,-48.094,-179.069,5.838,148.761
C00644=1196.291,71.629,-48.111,-179.066,5.839,148.760
C00645=1196.286,71.879,-48.128,-179.064,5.840,148.760
C00646=1196.282,72.128,-48.146,-179.061,5.841,148.759
C00647=1196.277,72.377,-48.162,-179.059,5.842,148.758
C00648=1196.271,72.627,-48.179,-179.056,5.843,148.758
C00649=1196.266,72.876,-48.197,-179.053,5.844,148.757
C00650=1196.262,73.125,-48.214,-179.051,5.844,148.757
C00651=1196.257,73.375,-48.231,-179.048,5.846,148.756
C00652=1196.252,73.624,-48.248,-179.046,5.847,148.756
C00653=1196.247,73.874,-48.266,-179.043,5.847,148.755
C00654=1196.242,74.122,-48.282,-179.041,5.848,148.754
C00655=1196.237,74.372,-48.300,-179.038,5.850,148.754
C00656=1196.232,74.621,-48.318,-179.035,5.850,148.753
C00657=1196.228,74.871,-48.334,-179.033,5.851,148.753
C00658=1196.222,75.121,-48.351,-179.030,5.852,148.752
C00659=1196.217,75.370,-48.369,-179.027,5.853,148.751
C00660=1196.213,75.619,-48.386,-179.025,5.854,148.751
C00661=1196.208,75.869,-48.404,-179.023,5.854,148.750
C00662=1196.202,76.118,-48.421,-179.020,5.856,148.750
C00663=1196.198,76.366,-48.438,-179.017,5.857,148.749
C00664=1196.193,76.616,-48.456,-179.015,5.857,148.749
C00665=1196.188,76.866,-48.473,-179.012,5.859,148.748
C00666=1196.183,77.115,-48.490,-179.009,5.859,148.748
C00667=1196.178,77.365,-48.508,-179.007,5.860,148.747
C00668=1196.173,77.614,-48.526,-179.004,5.861,148.746
C00669=1196.169,77.863,-48.542,-179.001,5.862,148.746
C00670=1196.164,78.113,-48.560,-178.999,5.863,148.745
C00671=1196.159,78.362,-48.577,-178.997,5.864,148.745
C00672=1196.154,78.611,-48.594,-178.994,5.866,148.744
C00673=1196.149,78.860,-48.612,-178.991,5.866,148.744
C00674=1196.144,79.109,-48.630,-178.989,5.867,148.743
C00675=1196.139,79.359,-48.647,-178.986,5.868,148.743
C00676=1196.134,79.608,-48.664,-178.983,5.869,148.742
C00677=1196.129,79.858,-48.682,-178.981,5.870,148.741
C00678=1196.124,80.107,-48.700,-178.978,5.870,148.741
C00679=1196.119,80.356,-48.718,-178.976,5.872,148.740
C00680=1196.115,80.625,-48.736,-178.973,5.873,148.740
C00681=1196.109,80.894,-48.754,-178.970,5.874,148.739
C00682=1196.104,81.161,-48.773,-178.967,5.875,148.738
C00683=1196.098,81.430,-48.792,-178.964,5.876,148.738
C00684=1196.093,81.679,-48.810,-178.962,5.877,148.737
C00685=1196.088,81.928,-48.828,-178.959,5.877,148.737
C00686=1196.084,82.178,-48.845,-178.957,5.879,148.736
C00687=1196.079,82.427,-48.863,-178.954,5.880,148.736
C00688=1196.074,82.676,-48.881,-178.952,5.881,148.735
C00689=1196.069,82.926,-48.898,-178.949,5.882,148.735
C00690=1196.064,83.175,-48.916,-178.946,5.883,148.734
C00691=1196.059,83.424,-48.934,-178.944,5.883,148.734
C00692=1196.055,83.674,-48.951,-178.941,5.885,148.733
C00693=1196.050,83.923,-48.969,-178.939,5.886,148.732
C00694=1196.045,84.172,-48.987,-178.936,5.886,148.732
C00695=1196.040,84.421,-49.005,-178.933,5.888,148.731
C00696=1196.035,84.671,-49.022,-178.931,5.889,148.731
C00697=1196.030,84.920,-49.040,-178.928,5.890,148.730
C00698=1196.025,85.170,-49.058,-178.925,5.891,148.730
C00699=1196.020,85.419,-49.076,-178.923,5.891,148.729
C00700=1196.016,85.669,-49.093,-178.920,5.892,148.729
C00701=1196.011,85.918,-49.111,-178.917,5.894,148.728
C00702=1196.006,86.167,-49.129,-178.915,5.895,148.727
C00703=1196.001,86.417,-49.147,-178.912,5.895,148.727
C00704=1195.996,86.666,-49.164,-178.910,5.897,148.726
C00705=1195.991,86.916,-49.182,-178.907,5.898,148.726
C00706=1195.986,87.165,-49.200,-178.904,5.899,148.725
C00707=1195.981,87.414,-49.218,-178.902,5.900,148.725
C00708=1195.976,87.663,-49.236,-178.899,5.900,148.724
C00709=1195.972,87.912,-49.254,-178.896,5.902,148.724
C00710=1195.967,88.161,-49.272,-178.894,5.903,148.723
C00711=1195.961,88.411,-49.289,-178.892,5.904,148.723
C00712=1195.956,88.660,-49.307,-178.889,5.905,148.722
C00713=1195.952,88.910,-49.325,-178.886,5.906,148.721
C00714=1195.947,89.159,-49.343,-178.884,5.906,148.721
C00715=1195.942,89.409,-49.361,-178.881,5.908,148.720
C00716=1195.937,89.658,-49.379,-178.878,5.909,148.720
C00717=1195.933,89.907,-49.397,-178.876,5.911,148.719
C00718=1195.928,90.156,-49.415,-178.873,5.911,148.719
C00719=1195.923,90.405,-49.433,-178.871,5.912,148.718
C00720=1195.918,90.654,-49.451,-178.868,5.913,148.718
C00721=1195.913,90.904,-49.469,-178.866,5.914,148.717
C00722=1195.909,91.154,-49.488,-178.863,5.915,148.717
C00723=1195.904,91.403,-49.506,-178.860,5.916,148.716
C00724=1195.899,91.652,-49.524,-178.858,5.917,148.715
C00725=1195.894,91.901,-49.542,-178.854,5.919,148.715
C00726=1195.889,92.150,-49.560,-178.852,5.919,148.714
C00727=1195.884,92.399,-49.577,-178.850,5.920,148.714
C00728=1195.880,92.649,-49.596,-178.847,5.922,148.713
C00729=1195.875,92.898,-49.614,-178.844,5.922,148.713
C00730=1195.870,93.148,-49.632,-178.842,5.923,148.712
C00731=1195.864,93.397,-49.650,-178.839,5.925,148.712
C00732=1195.859,93.646,-49.668,-178.837,5.926,148.711
C00733=1195.854,93.895,-49.686,-178.834,5.927,148.711
C00734=1195.850,94.145,-49.705,-178.832,5.928,148.710
C00735=1195.845,94.395,-49.723,-178.829,5.928,148.710
C00736=1195.840,94.644,-49.741,-178.826,5.930,148.709
C00737=1195.835,94.893,-49.759,-178.824,5.931,148.708
C00738=1195.831,95.141,-49.777,-178.821,5.932,148.708
C00739=1195.826,95.392,-49.796,-178.818,5.933,148.707
C00740=1195.821,95.641,-49.814,-178.816,5.934,148.707
C00741=1195.816,95.890,-49.832,-178.813,5.935,148.706
C00742=1195.811,96.139,-49.850,-178.811,5.936,148.706
C00743=1195.806,96.388,-49.868,-178.808,5.938,148.705
C00744=1195.802,96.638,-49.887,-178.806,5.939,148.705
C00745=1195.796,96.887,-49.906,-178.803,5.939,148.704
C00746=1195.791,97.136,-49.924,-178.800,5.941,148.704
C00747=1195.787,97.385,-49.942,-178.798,5.941,148.703
C00748=1195.782,97.635,-49.960,-178.795,5.943,148.703
C00749=1195.777,97.884,-49.979,-178.792,5.944,148.702
C00750=1195.772,98.133,-49.997,-178.790,5.946,148.702
C00751=1195.767,98.382,-50.015,-178.787,5.946,148.701
C00752=1195.763,98.632,-50.034,-178.785,5.947,148.701
C00753=1195.758,98.881,-50.052,-178.782,5.948,148.700
C00754=1195.753,99.130,-50.071,-178.780,5.949,148.700
C00755=1195.748,99.380,-50.089,-178.776,5.951,148.699
C00756=1195.743,99.629,-50.107,-178.774,5.952,148.699
C00757=1195.738,99.878,-50.127,-178.771,5.953,148.698
C00758=1195.733,100.128,-50.145,-178.769,5.954,148.697
C00759=1195.729,100.377,-50.163,-178.766,5.955,148.697
C00760=1195.724,100.626,-50.182,-178.764,5.956,148.696
C00761=1195.718,100.875,-50.200,-178.761,5.957,148.696
C00762=1195.714,101.125,-50.219,-178.758,5.959,148.695
C00763=1195.710,101.374,-50.237,-178.756,5.959,148.695
C00764=1195.704,101.623,-50.256,-178.753,5.961,148.694
C00765=1195.700,101.873,-50.275,-178.750,5.961,148.694
C00766=1195.695,102.122,-50.293,-178.748,5.962,148.693
C00767=1195.689,102.371,-50.311,-178.745,5.964,148.693
C00768=1195.685,102.621,-50.330,-178.743,5.965,148.692
C00769=1195.680,102.870,-50.348,-178.740,5.966,148.692
C00770=1195.675,103.119,-50.368,-178.737,5.967,148.691
C00771=1195.671,103.368,-50.386,-178.735,5.969,148.691
C00772=1195.666,103.617,-50.405,-178.732,5.969,148.690
C00773=1195.661,103.866,-50.423,-178.729,5.971,148.690
C00774=1195.656,104.116,-50.442,-178.727,5.972,148.689
C00775=1195.651,104.365,-50.461,-178.724,5.973,148.689
C00776=1195.646,104.614,-50.479,-178.722,5.974,148.688
C00777=1195.642,104.864,-50.498,-178.719,5.975,148.688
C00778=1195.636,105.113,-50.517,-178.716,5.976,148.687
C00779=1195.632,105.362,-50.536,-178.714,5.977,148.686
C00780=1195.627,105.611,-50.555,-178.711,5.979,148.686
C00781=1195.622,105.860,-50.573,-178.709,5.980,148.685
C00782=1195.618,106.110,-50.592,-178.706,5.981,148.685
C00783=1195.612,106.359,-50.611,-178.703,5.982,148.684
C00784=1195.607,106.627,-50.631,-178.700,5.983,148.684
C00785=1195.602,106.896,-50.651,-178.698,5.985,148.683
C00786=1195.597,107.164,-50.672,-178.695,5.986,148.683
C00787=1195.592,107.433,-50.692,-178.692,5.987,148.682
C00788=1195.587,107.682,-50.711,-178.690,5.988,148.682
C00789=1195.582,107.931,-50.729,-178.687,5.990,148.681
C00790=1195.577,108.181,-50.749,-178.684,5.990,148.681
C00791=1195.573,108.429,-50.767,-178.682,5.992,148.680
C00792=1195.568,108.679,-50.786,-178.679,5.993,148.680
C00793=1195.563,108.928,-50.805,-178.676,5.994,148.679
C00794=1195.558,109.177,-50.825,-178.674,5.995,148.679
C00795=1195.553,109.427,-50.843,-178.671,5.997,148.678
C00796=1195.548,109.676,-50.862,-178.669,5.998,148.678
C00797=1195.543,109.925,-50.881,-178.666,5.999,148.677
C00798=1195.538,110.174,-50.899,-178.664,6.000,148.677
C00799=1195.534,110.424,-50.919,-178.660,6.001,148.676
C00800=1195.529,110.672,-50.938,-178.658,6.002,148.676
C00801=1195.524,110.922,-50.957,-178.655,6.004,148.675
C00802=1195.519,111.171,-50.975,-178.653,6.005,148.675
C00803=1195.515,111.421,-50.995,-178.650,6.006,148.674
C00804=1195.509,111.670,-51.014,-178.648,6.007,148.674
C00805=1195.505,111.919,-51.033,-178.645,6.009,148.673
C00806=1195.500,112.168,-51.052,-178.642,6.009,148.673
C00807=1195.496,112.418,-51.071,-178.640,6.011,148.672
C00808=1195.490,112.666,-51.090,-178.637,6.012,148.671
C00809=1195.486,112.916,-51.110,-178.634,6.013,148.671
C00810=1195.481,113.165,-51.129,-178.632,6.014,148.671
C00811=1195.476,113.415,-51.148,-178.629,6.016,148.670
C00812=1195.471,113.664,-51.167,-178.627,6.017,148.670
C00813=1195.467,113.913,-51.186,-178.624,6.018,148.669
C00814=1195.461,114.162,-51.205,-178.622,6.019,148.669
C00815=1195.457,114.411,-51.225,-178.619,6.021,148.668
C00816=1195.452,114.660,-51.244,-178.616,6.021,148.668
C00817=1195.447,114.909,-51.263,-178.614,6.023,148.667
C00818=1195.442,115.159,-51.283,-178.611,6.024,148.666
C00819=1195.438,115.408,-51.301,-178.608,6.025,148.666
C00820=1195.433,115.658,-51.321,-178.606,6.026,148.666
C00821=1195.427,115.907,-51.340,-178.603,6.028,148.665
C00822=1195.423,116.156,-51.359,-178.600,6.029,148.665
C00823=1195.418,116.405,-51.378,-178.598,6.030,148.664
C00824=1195.413,116.654,-51.398,-178.595,6.032,148.664
C00825=1195.408,116.903,-51.417,-178.593,6.033,148.663
C00826=1195.404,117.152,-51.436,-178.590,6.034,148.663
C00827=1195.399,117.402,-51.456,-178.587,6.035,148.662
C00828=1195.394,117.651,-51.475,-178.584,6.037,148.662
C00829=1195.389,117.900,-51.495,-178.582,6.037,148.661
C00830=1195.385,118.149,-51.514,-178.579,6.039,148.661
C00831=1195.380,118.399,-51.533,-178.577,6.040,148.660
C00832=1195.375,118.648,-51.553,-178.574,6.042,148.660
C00833=1195.370,118.897,-51.572,-178.571,6.043,148.659
C00834=1195.366,119.146,-51.591,-178.569,6.044,148.659
C00835=1195.361,119.396,-51.611,-178.566,6.046,148.658
C00836=1195.356,119.645,-51.630,-178.564,6.046,148.658
C00837=1195.351,119.894,-51.650,-178.561,6.048,148.657
C00838=1195.346,120.143,-51.670,-178.558,6.049,148.657
C00839=1195.342,120.392,-51.689,-178.556,6.050,148.656
C00840=1195.337,120.641,-51.709,-178.553,6.051,148.656
C00841=1195.332,120.890,-51.728,-178.550,6.053,148.655
C00842=1195.327,121.140,-51.747,-178.548,6.054,148.655
C00843=1195.322,121.389,-51.767,-178.545,6.055,148.654
C00844=1195.317,121.638,-51.786,-178.542,6.057,148.654
C00845=1195.313,121.887,-51.807,-178.540,6.058,148.653
C00846=1195.309,122.136,-51.826,-178.537,6.059,148.653
C00847=1195.303,122.385,-51.845,-178.535,6.060,148.652
C00848=1195.298,122.635,-51.865,-178.532,6.062,148.652
C00849=1195.294,122.884,-51.884,-178.529,6.063,148.651
C00850=1195.289,123.133,-51.904,-178.527,6.064,148.651
C00851=1195.284,123.382,-51.924,-178.524,6.066,148.650
C00852=1195.279,123.632,-51.944,-178.521,6.067,148.650
C00853=1195.274,123.881,-51.963,-178.519,6.068,148.649
C00854=1195.269,124.130,-51.983,-178.517,6.069,148.649
C00855=1195.265,124.379,-52.003,-178.513,6.071,148.648
C00856=1195.261,124.628,-52.022,-178.511,6.072,148.648
C00857=1195.255,124.877,-52.041,-178.509,6.073,148.648
C00858=1195.251,125.126,-52.062,-178.506,6.075,148.647
C00859=1195.246,125.376,-52.081,-178.503,6.076,148.647
C00860=1195.241,125.625,-52.101,-178.501,6.077,148.646
C00861=1195.236,125.874,-52.121,-178.498,6.079,148.646
C00862=1195.232,126.123,-52.141,-178.495,6.080,148.645
C00863=1195.227,126.373,-52.160,-178.493,6.082,148.645
C00864=1195.222,126.622,-52.181,-178.490,6.082,148.644
C00865=1195.217,126.871,-52.200,-178.487,6.084,148.644
C00866=1195.213,127.120,-52.220,-178.484,6.085,148.643
C00867=1195.208,127.369,-52.240,-178.482,6.086,148.643
C00868=1195.203,127.619,-52.260,-178.479,6.088,148.642
C00869=1195.198,127.867,-52.280,-178.477,6.089,148.642
C00870=1195.193,128.116,-52.299,-178.474,6.090,148.641
C00871=1195.189,128.365,-52.320,-178.471,6.092,148.641
C00872=1195.184,128.615,-52.339,-178.469,6.093,148.640
C00873=1195.180,128.864,-52.360,-178.466,6.095,148.640
C00874=1195.174,129.113,-52.379,-178.464,6.095,148.639
C00875=1195.169,129.363,-52.399,-178.461,6.097,148.639
C00876=1195.164,129.612,-52.420,-178.458,6.099,148.638
C00877=1195.160,129.861,-52.439,-178.456,6.100,148.638
C00878=1195.155,130.110,-52.460,-178.453,6.101,148.638
C00879=1195.150,130.359,-52.479,-178.451,6.102,148.637
C00880=1195.146,130.608,-52.499,-178.448,6.104,148.637
C00881=1195.141,130.858,-52.519,-178.445,6.105,148.636
C00882=1195.136,131.107,-52.539,-178.443,6.106,148.636
C00883=1195.132,131.355,-52.560,-178.440,6.108,148.635
C00884=1195.126,131.605,-52.580,-178.437,6.110,148.635
C00885=1195.121,131.854,-52.600,-178.435,6.110,148.634
C00886=1195.117,132.103,-52.620,-178.432,6.112,148.634
C00887=1195.112,132.352,-52.640,-178.429,6.114,148.633
C00888=1195.107,132.621,-52.661,-178.427,6.114,148.633
C00889=1195.102,132.889,-52.684,-178.424,6.116,148.632
C00890=1195.096,133.158,-52.705,-178.421,6.118,148.632
C00891=1195.092,133.426,-52.727,-178.418,6.119,148.631
C00892=1195.087,133.676,-52.747,-178.416,6.121,148.631
C00893=1195.082,133.925,-52.767,-178.413,6.122,148.630
C00894=1195.077,134.174,-52.787,-178.410,6.123,148.630
C00895=1195.073,134.423,-52.808,-178.408,6.124,148.630
C00896=1195.068,134.672,-52.828,-178.405,6.126,148.629
C00897=1195.064,134.921,-52.848,-178.402,6.128,148.629
C00898=1195.058,135.171,-52.868,-178.400,6.129,148.628
C00899=1195.053,135.419,-52.889,-178.397,6.130,148.628
C00900=1195.049,135.668,-52.909,-178.394,6.132,148.627
C00901=1195.044,135.918,-52.929,-178.392,6.133,148.627
C00902=1195.039,136.167,-52.950,-178.389,6.134,148.626
C00903=1195.034,136.416,-52.970,-178.386,6.136,148.626
C00904=1195.030,136.665,-52.990,-178.384,6.137,148.625
C00905=1195.025,136.915,-53.010,-178.381,6.139,148.625
C00906=1195.020,137.164,-53.031,-178.378,6.140,148.624
C00907=1195.016,137.413,-53.051,-178.376,6.141,148.624
C00908=1195.011,137.662,-53.072,-178.373,6.143,148.624
C00909=1195.006,137.911,-53.093,-178.371,6.144,148.623
C00910=1195.002,138.160,-53.113,-178.368,6.145,148.623
C00911=1194.997,138.410,-53.133,-178.366,6.147,148.622
C00912=1194.992,138.659,-53.154,-178.363,6.149,148.622
C00913=1194.987,138.908,-53.174,-178.361,6.150,148.621
C00914=1194.982,139.156,-53.194,-178.358,6.151,148.621
C00915=1194.977,139.405,-53.215,-178.355,6.153,148.620
C00916=1194.973,139.654,-53.236,-178.353,6.154,148.620
C00917=1194.968,139.903,-53.256,-178.350,6.155,148.620
C00918=1194.963,140.152,-53.277,-178.347,6.157,148.619
C00919=1194.958,140.402,-53.297,-178.344,6.159,148.619
C00920=1194.954,140.651,-53.317,-178.342,6.160,148.618
C00921=1194.949,140.900,-53.338,-178.339,6.161,148.618
C00922=1194.944,141.149,-53.358,-178.336,6.163,148.617
C00923=1194.939,141.398,-53.379,-178.334,6.164,148.617
C00924=1194.935,141.647,-53.400,-178.331,6.166,148.617
C00925=1194.930,141.896,-53.420,-178.328,6.167,148.616
C00926=1194.926,142.146,-53.441,-178.326,6.168,148.616
C00927=1194.921,142.395,-53.462,-178.323,6.170,148.615
C00928=1194.916,142.645,-53.483,-178.321,6.171,148.615
C00929=1194.911,142.894,-53.503,-178.318,6.172,148.614
C00930=1194.906,143.143,-53.524,-178.315,6.174,148.614
C00931=1194.902,143.392,-53.544,-178.313,6.176,148.613
C00932=1194.897,143.641,-53.565,-178.310,6.177,148.613
C00933=1194.892,143.890,-53.586,-178.308,6.178,148.613
C00934=1194.888,144.138,-53.607,-178.305,6.180,148.612
C00935=1194.883,144.388,-53.628,-178.302,6.182,148.612
C00936=1194.878,144.636,-53.648,-178.300,6.182,148.611
C00937=1194.873,144.886,-53.669,-178.297,6.184,148.611
C00938=1194.869,145.135,-53.689,-178.294,6.186,148.610
C00939=1194.864,145.384,-53.710,-178.292,6.187,148.610
C00940=1194.859,145.633,-53.731,-178.289,6.188,148.609
C00941=1194.854,145.882,-53.752,-178.287,6.190,148.609
C00942=1194.850,146.131,-53.774,-178.284,6.192,148.608
C00943=1194.845,146.380,-53.794,-178.281,6.193,148.608
C00944=1194.840,146.630,-53.815,-178.279,6.194,148.608
C00945=1194.836,146.879,-53.835,-178.276,6.196,148.607
C00946=1194.831,147.128,-53.856,-178.273,6.198,148.607
C00947=1194.826,147.377,-53.877,-178.271,6.199,148.606
C00948=1194.821,147.625,-53.899,-178.268,6.200,148.606
C00949=1194.817,147.874,-53.919,-178.265,6.202,148.606
C00950=1194.812,148.124,-53.940,-178.263,6.204,148.605
C00951=1194.807,148.374,-53.961,-178.261,6.205,148.605
C00952=1194.803,148.622,-53.982,-178.257,6.206,148.604
C00953=1194.798,148.871,-54.003,-178.255,6.208,148.604
C00954=1194.793,149.121,-54.024,-178.252,6.210,148.603
C00955=1194.788,149.369,-54.045,-178.250,6.211,148.603
C00956=1194.783,149.618,-54.066,-178.247,6.212,148.602
C00957=1194.779,149.868,-54.087,-178.244,6.214,148.602
C00958=1194.774,150.117,-54.108,-178.241,6.216,148.602
C00959=1194.769,150.366,-54.130,-178.239,6.217,148.601
C00960=1194.765,150.615,-54.150,-178.237,6.218,148.601
C00961=1194.760,150.864,-54.171,-178.234,6.220,148.600
C00962=1194.755,151.112,-54.193,-178.231,6.222,148.600
C00963=1194.751,151.362,-54.213,-178.229,6.223,148.599
C00964=1194.746,151.611,-54.235,-178.226,6.224,148.599
C00965=1194.741,151.860,-54.256,-178.223,6.226,148.599
C00966=1194.736,152.109,-54.277,-178.221,6.228,148.598
C00967=1194.732,152.358,-54.298,-178.218,6.229,148.598
C00968=1194.727,152.608,-54.319,-178.215,6.230,148.597
C00969=1194.722,152.856,-54.341,-178.213,6.232,148.597
C00970=1194.718,153.105,-54.362,-178.210,6.234,148.597
C00971=1194.713,153.354,-54.383,-178.207,6.236,148.596
C00972=1194.708,153.603,-54.404,-178.205,6.236,148.596
C00973=1194.704,153.852,-54.426,-178.202,6.238,148.595
C00974=1194.698,154.102,-54.447,-178.199,6.240,148.595
C00975=1194.694,154.350,-54.468,-178.197,6.242,148.594
C00976=1194.689,154.599,-54.489,-178.195,6.243,148.594
C00977=1194.685,154.849,-54.511,-178.192,6.244,148.594
C00978=1194.680,155.098,-54.532,-178.189,6.246,148.593
C00979=1194.676,155.346,-54.553,-178.186,6.248,148.593
C00980=1194.670,155.595,-54.574,-178.183,6.249,148.592
C00981=1194.666,155.845,-54.596,-178.181,6.250,148.592
C00982=1194.661,156.094,-54.617,-178.179,6.252,148.592
C00983=1194.656,156.343,-54.639,-178.176,6.254,148.591
C00984=1194.652,156.592,-54.661,-178.173,6.256,148.591
C00985=1194.647,156.841,-54.681,-178.170,6.257,148.590
C00986=1194.642,157.090,-54.703,-178.168,6.258,148.590
C00987=1194.637,157.339,-54.724,-178.165,6.260,148.589
C00988=1194.633,157.588,-54.746,-178.163,6.262,148.589
C00989=1194.628,157.837,-54.768,-178.160,6.263,148.589
C00990=1194.623,158.086,-54.789,-178.157,6.265,148.588
C00991=1194.619,158.335,-54.811,-178.155,6.266,148.588
C00992=1194.614,158.605,-54.834,-178.152,6.268,148.587
C00993=1194.609,158.873,-54.858,-178.149,6.269,148.587
C00994=1194.604,159.142,-54.880,-178.147,6.271,148.587
C00995=1194.598,159.411,-54.903,-178.143,6.273,148.586
C00996=1194.594,159.660,-54.925,-178.141,6.274,148.586
C00997=1194.589,159.909,-54.947,-178.138,6.276,148.585
C00998=1194.584,160.159,-54.968,-178.135,6.278,148.585
C00999=1194.580,160.407,-54.990,-178.133,6.280,148.585
C01000=1194.575,160.656,-55.011,-178.130,6.282,148.584
C01001=1194.571,160.905,-55.033,-178.128,6.282,148.584
C01002=1194.566,161.154,-55.054,-178.125,6.284,148.583
C01003=1194.561,161.403,-55.076,-178.122,6.286,148.583
C01004=1194.557,161.652,-55.098,-178.119,6.288,148.582
C01005=1194.552,161.901,-55.120,-178.117,6.289,148.582
C01006=1194.547,162.150,-55.141,-178.114,6.291,148.582
C01007=1194.543,162.399,-55.163,-178.112,6.292,148.581
C01008=1194.537,162.648,-55.184,-178.109,6.294,148.581
C01009=1194.533,162.898,-55.206,-178.106,6.295,148.580
C01010=1194.528,163.146,-55.228,-178.104,6.297,148.580
C01011=1194.524,163.396,-55.250,-178.101,6.299,148.580
C01012=1194.519,163.644,-55.272,-178.098,6.301,148.579
C01013=1194.514,163.893,-55.293,-178.096,6.302,148.579
C01014=1194.510,164.142,-55.316,-178.093,6.303,148.578
C01015=1194.504,164.391,-55.338,-178.091,6.305,148.578
C01016=1194.500,164.641,-55.360,-178.088,6.307,148.578
C01017=1194.495,164.889,-55.382,-178.085,6.309,148.577
C01018=1194.491,165.139,-55.404,-178.082,6.310,148.577
C01019=1194.486,165.387,-55.425,-178.080,6.311,148.576
C01020=1194.481,165.636,-55.446,-178.077,6.313,148.576
C01021=1194.477,165.886,-55.468,-178.075,6.315,148.576
C01022=1194.472,166.134,-55.490,-178.072,6.317,148.575
C01023=1194.468,166.383,-55.513,-178.069,6.318,148.575
C01024=1194.463,166.632,-55.534,-178.067,6.320,148.575
C01025=1194.459,166.881,-55.556,-178.064,6.322,148.574
C01026=1194.453,167.130,-55.579,-178.061,6.324,148.574
C01027=1194.449,167.379,-55.601,-178.059,6.325,148.573
C01028=1194.444,167.628,-55.622,-178.057,6.326,148.573
C01029=1194.440,167.877,-55.645,-178.053,6.328,148.572
C01030=1194.435,168.126,-55.666,-178.051,6.330,148.572
C01031=1194.431,168.375,-55.688,-178.048,6.331,148.572
C01032=1194.425,168.624,-55.711,-178.045,6.333,148.571
C01033=1194.421,168.874,-55.733,-178.043,6.335,148.571
C01034=1194.416,169.122,-55.754,-178.040,6.337,148.571
C01035=1194.412,169.372,-55.776,-178.038,6.338,148.570
C01036=1194.407,169.620,-55.799,-178.035,6.340,148.570
C01037=1194.402,169.869,-55.821,-178.033,6.341,148.570
C01038=1194.397,170.118,-55.843,-178.030,6.343,148.569
C01039=1194.393,170.367,-55.865,-178.027,6.345,148.569
C01040=1194.388,170.616,-55.887,-178.025,6.347,148.568
C01041=1194.383,170.865,-55.910,-178.022,6.349,148.568
C01042=1194.378,171.114,-55.932,-178.019,6.350,148.568
C01043=1194.374,171.363,-55.954,-178.017,6.351,148.567
C01044=1194.370,171.612,-55.976,-178.014,6.353,148.567
C01045=1194.364,171.861,-55.998,-178.011,6.355,148.566
C01046=1194.360,172.110,-56.021,-178.009,6.356,148.566
C01047=1194.356,172.359,-56.043,-178.006,6.358,148.566
C01048=1194.350,172.608,-56.065,-178.003,6.360,148.565
C01049=1194.346,172.856,-56.088,-178.001,6.362,148.565
C01050=1194.342,173.106,-56.110,-177.998,6.363,148.565
C01051=1194.337,173.355,-56.132,-177.995,6.365,148.564
C01052=1194.332,173.603,-56.155,-177.993,6.367,148.564
C01053=1194.328,173.853,-56.177,-177.990,6.369,148.563
C01054=1194.322,174.102,-56.199,-177.988,6.370,148.563
C01055=1194.318,174.350,-56.222,-177.985,6.372,148.563
C01056=1194.314,174.600,-56.244,-177.983,6.373,148.562
C01057=1194.308,174.849,-56.266,-177.980,6.375,148.562
C01058=1194.304,175.097,-56.289,-177.977,6.377,148.562
C01059=1194.300,175.346,-56.311,-177.975,6.379,148.561
C01060=1194.295,175.595,-56.334,-177.972,6.381,148.561
C01061=1194.291,175.844,-56.356,-177.969,6.382,148.561
C01062=1194.285,176.093,-56.378,-177.967,6.384,148.560
C01063=1194.281,176.342,-56.401,-177.964,6.386,148.560
C01064=1194.277,176.591,-56.423,-177.961,6.388,148.559
C01065=1194.271,176.840,-56.446,-177.959,6.390,148.559
C01066=1194.267,177.089,-56.468,-177.956,6.391,148.559
C01067=1194.262,177.338,-56.492,-177.954,6.392,148.558
C01068=1194.258,177.587,-56.513,-177.951,6.394,148.558
C01069=1194.253,177.836,-56.537,-177.948,6.396,148.558
C01070=1194.249,178.085,-56.559,-177.946,6.398,148.557
C01071=1194.244,178.333,-56.581,-177.943,6.400,148.557
C01072=1194.239,178.583,-56.604,-177.940,6.401,148.557
C01073=1194.235,178.831,-56.626,-177.937,6.403,148.556
C01074=1194.230,179.080,-56.649,-177.935,6.405,148.556
C01075=1194.226,179.329,-56.671,-177.932,6.406,148.555
C01076=1194.221,179.578,-56.695,-177.929,6.408,148.555
C01077=1194.217,179.828,-56.717,-177.927,6.410,148.555
C01078=1194.211,180.076,-56.740,-177.924,6.412,148.554
C01079=1194.207,180.325,-56.762,-177.921,6.414,148.554
C01080=1194.202,180.574,-56.785,-177.919,6.415,148.553
C01081=1194.197,180.823,-56.808,-177.916,6.417,148.553
C01082=1194.193,181.072,-56.830,-177.913,6.419,148.553
C01083=1194.188,181.321,-56.854,-177.911,6.421,148.553
C01084=1194.184,181.570,-56.876,-177.908,6.423,148.552
C01085=1194.178,181.819,-56.899,-177.906,6.425,148.552
C01086=1194.175,182.067,-56.921,-177.903,6.426,148.552
C01087=1194.170,182.316,-56.945,-177.901,6.427,148.551
C01088=1194.166,182.565,-56.968,-177.898,6.429,148.551
C01089=1194.160,182.814,-56.990,-177.896,6.431,148.550
C01090=1194.156,183.063,-57.013,-177.893,6.433,148.550
C01091=1194.152,183.312,-57.036,-177.890,6.435,148.550
C01092=1194.147,183.561,-57.059,-177.888,6.436,148.549
C01093=1194.142,183.810,-57.082,-177.885,6.438,148.549
C01094=1194.137,184.058,-57.104,-177.882,6.440,148.549
C01095=1194.133,184.308,-57.128,-177.880,6.442,148.548
C01096=1194.128,184.577,-57.152,-177.876,6.444,148.548
C01097=1194.123,184.847,-57.177,-177.873,6.446,148.547
C01098=1194.117,185.117,-57.202,-177.871,6.448,148.547
C01099=1194.113,185.386,-57.227,-177.868,6.450,148.547
C01100=1194.108,185.635,-57.250,-177.865,6.451,148.546
C01101=1194.103,185.884,-57.273,-177.863,6.453,148.546
C01102=1194.099,186.133,-57.296,-177.860,6.455,148.546
C01103=1194.095,186.382,-57.320,-177.857,6.457,148.545
C01104=1194.089,186.630,-57.343,-177.855,6.459,148.545
C01105=1194.085,186.879,-57.365,-177.852,6.460,148.545
C01106=1194.080,187.128,-57.388,-177.850,6.462,148.544
C01107=1194.076,187.378,-57.411,-177.847,6.464,148.544
C01108=1194.071,187.627,-57.435,-177.844,6.466,148.544
C01109=1194.067,187.875,-57.457,-177.842,6.468,148.543
C01110=1194.062,188.124,-57.480,-177.839,6.470,148.543
C01111=1194.057,188.373,-57.504,-177.836,6.471,148.543
C01112=1194.052,188.622,-57.527,-177.834,6.473,148.542
C01113=1194.048,188.871,-57.550,-177.831,6.475,148.542
C01114=1194.044,189.119,-57.573,-177.829,6.477,148.542
C01115=1194.039,189.368,-57.597,-177.826,6.479,148.541
C01116=1194.034,189.617,-57.620,-177.823,6.480,148.541
C01117=1194.030,189.867,-57.643,-177.821,6.482,148.541
C01118=1194.025,190.116,-57.667,-177.818,6.484,148.540
C01119=1194.020,190.364,-57.689,-177.815,6.486,148.540
C01120=1194.016,190.613,-57.712,-177.813,6.488,148.540
C01121=1194.011,190.861,-57.737,-177.810,6.490,148.539
C01122=1194.007,191.110,-57.760,-177.808,6.492,148.539
C01123=1194.002,191.359,-57.783,-177.805,6.493,148.539
C01124=1193.997,191.608,-57.807,-177.802,6.495,148.538
C01125=1193.992,191.857,-57.830,-177.799,6.498,148.538
C01126=1193.989,192.106,-57.853,-177.796,6.500,148.538
C01127=1193.984,192.355,-57.876,-177.794,6.501,148.537
C01128=1193.979,192.604,-57.899,-177.791,6.503,148.537
C01129=1193.975,192.852,-57.924,-177.788,6.505,148.537
C01130=1193.970,193.101,-57.947,-177.786,6.507,148.536
C01131=1193.965,193.350,-57.970,-177.783,6.509,148.536
C01132=1193.961,193.599,-57.994,-177.781,6.511,148.536
C01133=1193.956,193.848,-58.017,-177.778,6.512,148.535
C01134=1193.952,194.097,-58.041,-177.776,6.514,148.535
C01135=1193.947,194.346,-58.064,-177.773,6.516,148.535
C01136=1193.942,194.595,-58.088,-177.770,6.518,148.534
C01137=1193.937,194.844,-58.111,-177.768,6.520,148.534
C01138=1193.933,195.092,-58.135,-177.765,6.522,148.534
C01139=1193.928,195.341,-58.159,-177.762,6.523,148.533
C01140=1193.924,195.590,-58.181,-177.760,6.525,148.533
C01141=1193.920,195.839,-58.205,-177.757,6.527,148.533
C01142=1193.915,196.088,-58.229,-177.754,6.529,148.532
C01143=1193.911,196.337,-58.252,-177.752,6.531,148.532
C01144=1193.905,196.585,-58.277,-177.750,6.533,148.532
C01145=1193.901,196.834,-58.300,-177.746,6.535,148.532
C01146=1193.896,197.083,-58.323,-177.744,6.537,148.531
C01147=1193.892,197.332,-58.348,-177.741,6.539,148.531
C01148=1193.887,197.581,-58.371,-177.738,6.541,148.530
C01149=1193.882,197.830,-58.394,-177.736,6.543,148.530
C01150=1193.878,198.078,-58.418,-177.733,6.545,148.530
C01151=1193.873,198.327,-58.442,-177.731,6.547,148.530
C01152=1193.869,198.576,-58.466,-177.728,6.548,148.529
C01153=1193.864,198.825,-58.489,-177.726,6.550,148.529
C01154=1193.860,199.073,-58.513,-177.723,6.552,148.529
C01155=1193.855,199.322,-58.537,-177.720,6.554,148.528
C01156=1193.851,199.571,-58.561,-177.718,6.556,148.528
C01157=1193.846,199.820,-58.584,-177.715,6.558,148.528
C01158=1193.842,200.068,-58.608,-177.712,6.560,148.527
C01159=1193.837,200.318,-58.632,-177.710,6.562,148.527
C01160=1193.832,200.567,-58.656,-177.707,6.564,148.527
C01161=1193.828,200.816,-58.680,-177.704,6.566,148.526
C01162=1193.823,201.064,-58.704,-177.702,6.568,148.526
C01163=1193.818,201.313,-58.727,-177.699,6.570,148.526
C01164=1193.814,201.561,-58.751,-177.696,6.571,148.525
C01165=1193.809,201.810,-58.775,-177.694,6.573,148.525
C01166=1193.804,202.059,-58.799,-177.691,6.575,148.525
C01167=1193.800,202.308,-58.823,-177.689,6.577,148.525
C01168=1193.796,202.557,-58.847,-177.686,6.580,148.524
C01169=1193.791,202.806,-58.871,-177.683,6.582,148.524
C01170=1193.787,203.055,-58.895,-177.680,6.583,148.524
C01171=1193.782,203.304,-58.919,-177.678,6.585,148.523
C01172=1193.777,203.552,-58.943,-177.675,6.587,148.523
C01173=1193.772,203.801,-58.967,-177.673,6.589,148.523
C01174=1193.769,204.050,-58.991,-177.670,6.591,148.522
C01175=1193.764,204.299,-59.016,-177.667,6.593,148.522
C01176=1193.759,204.547,-59.040,-177.665,6.595,148.522
C01177=1193.754,204.796,-59.063,-177.662,6.597,148.521
C01178=1193.750,205.045,-59.087,-177.659,6.599,148.521
C01179=1193.745,205.293,-59.112,-177.657,6.601,148.521
C01180=1193.741,205.543,-59.136,-177.654,6.603,148.521
C01181=1193.736,205.792,-59.160,-177.651,6.605,148.520
C01182=1193.732,206.040,-59.184,-177.649,6.607,148.520
C01183=1193.727,206.289,-59.209,-177.647,6.609,148.520
C01184=1193.722,206.537,-59.233,-177.644,6.611,148.520
C01185=1193.718,206.787,-59.256,-177.641,6.613,148.519
C01186=1193.713,207.036,-59.281,-177.638,6.615,148.519
C01187=1193.709,207.284,-59.305,-177.635,6.617,148.519
C01188=1193.704,207.532,-59.329,-177.633,6.619,148.518
C01189=1193.700,207.782,-59.354,-177.631,6.621,148.518
C01190=1193.696,208.030,-59.378,-177.628,6.623,148.518
C01191=1193.690,208.280,-59.402,-177.625,6.624,148.517
C01192=1193.686,208.528,-59.426,-177.622,6.627,148.517
C01193=1193.682,208.777,-59.451,-177.619,6.629,148.517
C01194=1193.677,209.026,-59.475,-177.617,6.631,148.517
C01195=1193.672,209.274,-59.499,-177.615,6.633,148.516
C01196=1193.668,209.523,-59.524,-177.612,6.635,148.516
C01197=1193.663,209.772,-59.549,-177.609,6.636,148.516
C01198=1193.659,210.020,-59.573,-177.606,6.639,148.515
C01199=1193.654,210.269,-59.597,-177.604,6.641,148.515
C01200=1193.649,210.539,-59.624,-177.601,6.643,148.515
C01201=1193.645,210.811,-59.650,-177.598,6.646,148.515
C01202=1193.640,211.081,-59.677,-177.595,6.648,148.514
C01203=1193.634,211.351,-59.703,-177.593,6.649,148.514
C01204=1193.629,211.600,-59.728,-177.589,6.652,148.514
C01205=1193.625,211.849,-59.752,-177.587,6.654,148.513
C01206=1193.620,212.097,-59.777,-177.585,6.656,148.513
C01207=1193.616,212.346,-59.801,-177.582,6.658,148.513
C01208=1193.611,212.595,-59.826,-177.579,6.660,148.512
C01209=1193.607,212.844,-59.850,-177.577,6.661,148.512
C01210=1193.602,213.092,-59.875,-177.574,6.664,148.512
C01211=1193.598,213.341,-59.900,-177.571,6.666,148.512
C01212=1193.593,213.590,-59.925,-177.569,6.668,148.511
C01213=1193.589,213.838,-59.949,-177.566,6.670,148.511
C01214=1193.584,214.087,-59.974,-177.563,6.672,148.511
C01215=1193.580,214.336,-59.998,-177.561,6.675,148.511
C01216=1193.575,214.585,-60.023,-177.558,6.676,148.510
C01217=1193.571,214.834,-60.047,-177.555,6.678,148.510
C01218=1193.566,215.082,-60.072,-177.553,6.680,148.510
C01219=1193.562,215.331,-60.097,-177.551,6.682,148.509
C01220=1193.557,215.580,-60.121,-177.547,6.685,148.509
C01221=1193.552,215.828,-60.146,-177.545,6.687,148.509
C01222=1193.548,216.077,-60.171,-177.542,6.689,148.508
C01223=1193.543,216.326,-60.196,-177.540,6.691,148.508
C01224=1193.539,216.575,-60.221,-177.537,6.692,148.508
C01225=1193.535,216.823,-60.245,-177.535,6.694,148.508
C01226=1193.530,217.071,-60.270,-177.531,6.697,148.507
C01227=1193.526,217.321,-60.295,-177.529,6.699,148.507
C01228=1193.521,217.569,-60.320,-177.526,6.701,148.507
C01229=1193.516,217.819,-60.345,-177.524,6.703,148.507
C01230=1193.512,218.067,-60.369,-177.521,6.706,148.507
C01231=1193.508,218.316,-60.394,-177.518,6.708,148.506
C01232=1193.503,218.565,-60.419,-177.516,6.709,148.506
C01233=1193.498,218.812,-60.444,-177.513,6.711,148.506
C01234=1193.494,219.062,-60.469,-177.511,6.713,148.505
C01235=1193.489,219.310,-60.494,-177.508,6.716,148.505
C01236=1193.485,219.559,-60.519,-177.505,6.718,148.505
C01237=1193.480,219.808,-60.543,-177.503,6.720,148.505
C01238=1193.476,220.057,-60.569,-177.500,6.722,148.504
C01239=1193.471,220.305,-60.594,-177.498,6.724,148.504
C01240=1193.467,220.554,-60.620,-177.494,6.726,148.504
C01241=1193.462,220.803,-60.644,-177.492,6.728,148.504
C01242=1193.458,221.051,-60.669,-177.490,6.730,148.503
C01243=1193.453,221.300,-60.694,-177.487,6.732,148.503
C01244=1193.449,221.549,-60.720,-177.484,6.735,148.503
C01245=1193.444,221.797,-60.744,-177.482,6.737,148.503
C01246=1193.440,222.046,-60.770,-177.479,6.739,148.502
C01247=1193.435,222.295,-60.794,-177.476,6.740,148.502
C01248=1193.431,222.544,-60.820,-177.474,6.743,148.502
C01249=1193.426,222.792,-60.845,-177.471,6.745,148.501
C01250=1193.422,223.041,-60.870,-177.468,6.747,148.501
C01251=1193.417,223.290,-60.895,-177.466,6.749,148.501
C01252=1193.413,223.538,-60.920,-177.463,6.751,148.501
C01253=1193.408,223.787,-60.946,-177.460,6.754,148.500
C01254=1193.403,224.036,-60.971,-177.458,6.756,148.500
C01255=1193.399,224.285,-60.997,-177.455,6.758,148.500
C01256=1193.395,224.533,-61.021,-177.453,6.760,148.500
C01257=1193.390,224.782,-61.046,-177.450,6.762,148.500
C01258=1193.386,225.030,-61.072,-177.447,6.764,148.499
C01259=1193.381,225.280,-61.097,-177.445,6.766,148.499
C01260=1193.376,225.528,-61.122,-177.443,6.768,148.499
C01261=1193.372,225.776,-61.148,-177.439,6.771,148.499
C01262=1193.368,226.026,-61.173,-177.437,6.773,148.498
C01263=1193.363,226.274,-61.198,-177.435,6.775,148.498
C01264=1193.358,226.523,-61.224,-177.432,6.777,148.498
C01265=1193.354,226.771,-61.249,-177.429,6.779,148.497
C01266=1193.349,227.020,-61.274,-177.427,6.782,148.497
C01267=1193.345,227.269,-61.300,-177.424,6.783,148.497
C01268=1193.341,227.517,-61.325,-177.422,6.786,148.497
C01269=1193.337,227.766,-61.351,-177.419,6.788,148.497
C01270=1193.331,228.014,-61.375,-177.416,6.790,148.496
C01271=1193.327,228.263,-61.401,-177.414,6.792,148.496
C01272=1193.323,228.512,-61.427,-177.411,6.794,148.496
C01273=1193.318,228.760,-61.452,-177.408,6.797,148.496
C01274=1193.314,229.009,-61.478,-177.406,6.799,148.495
C01275=1193.310,229.258,-61.504,-177.403,6.801,148.495
C01276=1193.305,229.506,-61.528,-177.400,6.803,148.495
C01277=1193.300,229.755,-61.554,-177.398,6.805,148.495
C01278=1193.295,230.004,-61.581,-177.395,6.807,148.494
C01279=1193.291,230.252,-61.606,-177.393,6.809,148.494
C01280=1193.286,230.501,-61.632,-177.390,6.812,148.494
C01281=1193.282,230.750,-61.657,-177.387,6.814,148.494
C01282=1193.277,230.998,-61.683,-177.385,6.816,148.494
C01283=1193.273,231.247,-61.709,-177.382,6.818,148.493
C01284=1193.269,231.496,-61.734,-177.380,6.821,148.493
C01285=1193.264,231.744,-61.760,-177.377,6.823,148.493
C01286=1193.260,231.993,-61.786,-177.374,6.825,148.493
C01287=1193.256,232.242,-61.811,-177.371,6.828,148.492
C01288=1193.251,232.490,-61.837,-177.369,6.829,148.492
C01289=1193.247,232.738,-61.862,-177.367,6.831,148.492
C01290=1193.242,232.988,-61.889,-177.364,6.833,148.492
C01291=1193.237,233.236,-61.914,-177.361,6.836,148.491
C01292=1193.233,233.484,-61.940,-177.359,6.838,148.491
C01293=1193.228,233.733,-61.966,-177.356,6.840,148.491
C01294=1193.224,233.982,-61.991,-177.353,6.843,148.491
C01295=1193.219,234.230,-62.017,-177.351,6.845,148.491
C01296=1193.214,234.479,-62.043,-177.349,6.847,148.490
C01297=1193.210,234.728,-62.069,-177.345,6.850,148.490
C01298=1193.206,234.977,-62.095,-177.343,6.851,148.490
C01299=1193.201,235.225,-62.120,-177.340,6.854,148.490
C01300=1193.197,235.473,-62.146,-177.337,6.856,148.489
C01301=1193.192,235.722,-62.173,-177.335,6.858,148.489
C01302=1193.188,235.971,-62.199,-177.332,6.860,148.489
C01303=1193.184,236.220,-62.224,-177.330,6.862,148.489
C01304=1193.178,236.491,-62.252,-177.327,6.865,148.489
C01305=1193.174,236.762,-62.281,-177.324,6.868,148.488
C01306=1193.169,237.035,-62.309,-177.321,6.870,148.488
C01307=1193.164,237.305,-62.338,-177.319,6.873,148.488
C01308=1193.159,237.554,-62.364,-177.316,6.874,148.488
C01309=1193.155,237.803,-62.389,-177.313,6.877,148.488
C01310=1193.150,238.051,-62.416,-177.311,6.879,148.487
C01311=1193.146,238.300,-62.442,-177.308,6.881,148.487
C01312=1193.142,238.549,-62.468,-177.305,6.884,148.487
C01313=1193.136,238.797,-62.494,-177.303,6.886,148.487
C01314=1193.133,239.045,-62.520,-177.300,6.888,148.487
C01315=1193.128,239.294,-62.546,-177.297,6.891,148.486
C01316=1193.123,239.543,-62.572,-177.295,6.893,148.486
C01317=1193.119,239.792,-62.599,-177.292,6.895,148.486
C01318=1193.115,240.040,-62.625,-177.290,6.898,148.486
C01319=1193.110,240.289,-62.651,-177.287,6.899,148.485
C01320=1193.106,240.537,-62.677,-177.285,6.902,148.485
C01321=1193.101,240.786,-62.703,-177.282,6.904,148.485
C01322=1193.097,241.034,-62.730,-177.279,6.906,148.485
C01323=1193.093,241.283,-62.756,-177.277,6.908,148.485
C01324=1193.088,241.532,-62.782,-177.274,6.911,148.485
C01325=1193.084,241.780,-62.808,-177.271,6.913,148.484
C01326=1193.080,242.029,-62.834,-177.269,6.915,148.484
C01327=1193.074,242.277,-62.861,-177.266,6.918,148.484
C01328=1193.070,242.526,-62.887,-177.264,6.920,148.484
C01329=1193.065,242.774,-62.914,-177.261,6.922,148.483
C01330=1193.061,243.023,-62.939,-177.259,6.925,148.483
C01331=1193.056,243.272,-62.966,-177.256,6.927,148.483
C01332=1193.052,243.520,-62.992,-177.253,6.930,148.483
C01333=1193.048,243.769,-63.019,-177.251,6.932,148.483
C01334=1193.043,244.018,-63.045,-177.248,6.934,148.483
C01335=1193.039,244.266,-63.072,-177.245,6.936,148.482
C01336=1193.035,244.514,-63.099,-177.243,6.939,148.482
C01337=1193.031,244.763,-63.124,-177.240,6.940,148.482
C01338=1193.026,245.012,-63.151,-177.238,6.943,148.482
C01339=1193.022,245.260,-63.177,-177.236,6.945,148.482
C01340=1193.017,245.509,-63.204,-177.232,6.948,148.481
C01341=1193.012,245.757,-63.231,-177.230,6.950,148.481
C01342=1193.008,246.006,-63.257,-177.228,6.952,148.481
C01343=1193.003,246.254,-63.284,-177.225,6.955,148.481
C01344=1192.999,246.502,-63.310,-177.222,6.957,148.481
C01345=1192.994,246.751,-63.337,-177.220,6.959,148.481
C01346=1192.990,247.000,-63.363,-177.217,6.962,148.480
C01347=1192.985,247.248,-63.390,-177.215,6.964,148.480
C01348=1192.981,247.497,-63.416,-177.211,6.967,148.480
C01349=1192.977,247.745,-63.443,-177.209,6.969,148.480
C01350=1192.972,247.994,-63.470,-177.207,6.971,148.480
C01351=1192.968,248.242,-63.496,-177.204,6.974,148.479
C01352=1192.963,248.491,-63.523,-177.202,6.976,148.479
C01353=1192.958,248.740,-63.550,-177.199,6.978,148.479
C01354=1192.955,248.989,-63.577,-177.196,6.981,148.479
C01355=1192.950,249.237,-63.604,-177.194,6.982,148.479
C01356=1192.946,249.485,-63.630,-177.191,6.985,148.479
C01357=1192.942,249.734,-63.656,-177.188,6.987,148.478
C01358=1192.937,249.983,-63.684,-177.186,6.990,148.478
C01359=1192.933,250.231,-63.710,-177.184,6.992,148.478
C01360=1192.928,250.480,-63.737,-177.180,6.995,148.478
C01361=1192.924,250.728,-63.764,-177.178,6.997,148.478
C01362=1192.919,250.976,-63.791,-177.176,6.999,148.477
C01363=1192.915,251.225,-63.818,-177.173,7.002,148.477
C01364=1192.910,251.473,-63.845,-177.171,7.004,148.477
C01365=1192.905,251.722,-63.871,-177.168,7.007,148.477
C01366=1192.902,251.970,-63.898,-177.165,7.009,148.477
C01367=1192.897,252.219,-63.925,-177.163,7.011,148.477
C01368=1192.892,252.467,-63.952,-177.160,7.014,148.477
C01369=1192.888,252.716,-63.979,-177.157,7.016,148.476
C01370=1192.884,252.965,-64.006,-177.155,7.019,148.476
C01371=1192.880,253.213,-64.033,-177.152,7.021,148.476
C01372=1192.875,253.462,-64.060,-177.149,7.024,148.476
C01373=1192.870,253.710,-64.087,-177.147,7.026,148.476
C01374=1192.866,253.959,-64.114,-177.145,7.028,148.476
C01375=1192.862,254.207,-64.140,-177.142,7.031,148.475
C01376=1192.857,254.456,-64.167,-177.140,7.033,148.475
C01377=1192.852,254.704,-64.194,-177.136,7.035,148.475
C01378=1192.849,254.953,-64.223,-177.134,7.038,148.475
C01379=1192.844,255.201,-64.250,-177.132,7.041,148.475
C01380=1192.840,255.449,-64.276,-177.129,7.042,148.475
C01381=1192.835,255.698,-64.303,-177.126,7.045,148.475
C01382=1192.831,255.946,-64.330,-177.124,7.048,148.474
C01383=1192.826,256.195,-64.357,-177.121,7.050,148.474
C01384=1192.822,256.444,-64.385,-177.119,7.052,148.474
C01385=1192.817,256.692,-64.412,-177.116,7.054,148.474
C01386=1192.813,256.940,-64.440,-177.113,7.057,148.474
C01387=1192.808,257.189,-64.467,-177.111,7.059,148.474
C01388=1192.804,257.437,-64.493,-177.108,7.062,148.473
C01389=1192.800,257.685,-64.520,-177.106,7.064,148.473
C01390=1192.796,257.935,-64.548,-177.103,7.067,148.473
C01391=1192.791,258.183,-64.575,-177.100,7.069,148.473
C01392=1192.787,258.431,-64.602,-177.098,7.072,148.473
C01393=1192.782,258.680,-64.629,-177.096,7.074,148.473
C01394=1192.778,258.929,-64.657,-177.092,7.077,148.473
C01395=1192.774,259.177,-64.685,-177.090,7.079,148.472
C01396=1192.769,259.425,-64.712,-177.088,7.082,148.472
C01397=1192.764,259.674,-64.739,-177.085,7.084,148.472
C01398=1192.760,259.921,-64.767,-177.082,7.087,148.472
C01399=1192.756,260.171,-64.794,-177.080,7.089,148.472
C01400=1192.751,260.419,-64.821,-177.077,7.092,148.472
C01401=1192.747,260.667,-64.849,-177.075,7.094,148.472
C01402=1192.742,260.916,-64.876,-177.073,7.096,148.471
C01403=1192.738,261.165,-64.903,-177.069,7.099,148.471
C01404=1192.734,261.413,-64.931,-177.067,7.101,148.471
C01405=1192.729,261.661,-64.958,-177.064,7.104,148.471
C01406=1192.725,261.910,-64.986,-177.062,7.106,148.471
C01407=1192.721,262.158,-65.013,-177.059,7.109,148.471
C01408=1192.716,262.431,-65.044,-177.056,7.112,148.471
C01409=1192.711,262.704,-65.074,-177.053,7.114,148.470
C01410=1192.706,262.976,-65.104,-177.050,7.117,148.470
C01411=1192.701,263.249,-65.134,-177.048,7.119,148.470
C01412=1192.697,263.498,-65.162,-177.045,7.122,148.470
C01413=1192.693,263.746,-65.190,-177.043,7.124,148.470
C01414=1192.688,263.995,-65.217,-177.040,7.127,148.470
C01415=1192.684,264.243,-65.245,-177.038,7.129,148.470
C01416=1192.679,264.492,-65.272,-177.035,7.132,148.470
C01417=1192.675,264.740,-65.300,-177.033,7.134,148.469
C01418=1192.671,264.988,-65.328,-177.030,7.137,148.469
C01419=1192.666,265.237,-65.355,-177.027,7.139,148.469
C01420=1192.662,265.485,-65.383,-177.025,7.142,148.469
C01421=1192.658,265.734,-65.411,-177.022,7.144,148.469
C01422=1192.653,265.982,-65.439,-177.019,7.147,148.469
C01423=1192.648,266.230,-65.467,-177.017,7.150,148.469
C01424=1192.644,266.479,-65.494,-177.014,7.152,148.469
C01425=1192.640,266.727,-65.522,-177.011,7.155,148.468
C01426=1192.636,266.976,-65.550,-177.009,7.157,148.468
C01427=1192.631,267.225,-65.578,-177.006,7.160,148.468
C01428=1192.626,267.472,-65.606,-177.004,7.162,148.468
C01429=1192.623,267.721,-65.634,-177.001,7.165,148.468
C01430=1192.618,267.970,-65.661,-176.999,7.167,148.468
C01431=1192.613,268.218,-65.689,-176.996,7.170,148.468
C01432=1192.609,268.466,-65.717,-176.994,7.172,148.468
C01433=1192.605,268.714,-65.745,-176.991,7.175,148.467
C01434=1192.601,268.963,-65.772,-176.989,7.177,148.467
C01435=1192.596,269.212,-65.801,-176.986,7.180,148.467
C01436=1192.592,269.460,-65.829,-176.983,7.183,148.467
C01437=1192.588,269.708,-65.857,-176.981,7.185,148.467
C01438=1192.582,269.956,-65.885,-176.978,7.188,148.467
C01439=1192.578,270.205,-65.913,-176.976,7.190,148.467
C01440=1192.574,270.453,-65.940,-176.973,7.193,148.467
C01441=1192.570,270.702,-65.969,-176.970,7.195,148.466
C01442=1192.565,270.950,-65.997,-176.968,7.198,148.466
C01443=1192.561,271.199,-66.025,-176.966,7.200,148.466
C01444=1192.556,271.447,-66.053,-176.963,7.203,148.466
C01445=1192.553,271.695,-66.081,-176.960,7.206,148.466
C01446=1192.548,271.943,-66.109,-176.958,7.208,148.466
C01447=1192.543,272.193,-66.137,-176.955,7.211,148.466
C01448=1192.539,272.441,-66.165,-176.953,7.213,148.466
C01449=1192.535,272.689,-66.193,-176.950,7.216,148.466
C01450=1192.530,272.937,-66.222,-176.948,7.218,148.466
C01451=1192.527,273.186,-66.250,-176.945,7.221,148.465
C01452=1192.521,273.434,-66.278,-176.942,7.224,148.465
C01453=1192.518,273.683,-66.306,-176.940,7.226,148.465
C01454=1192.513,273.931,-66.335,-176.937,7.229,148.465
C01455=1192.509,274.179,-66.363,-176.935,7.231,148.465
C01456=1192.504,274.427,-66.391,-176.932,7.234,148.465
C01457=1192.500,274.676,-66.419,-176.930,7.236,148.465
C01458=1192.496,274.924,-66.447,-176.927,7.239,148.465
C01459=1192.491,275.172,-66.477,-176.924,7.242,148.465
C01460=1192.487,275.420,-66.504,-176.922,7.244,148.465
C01461=1192.483,275.669,-66.533,-176.919,7.247,148.464
C01462=1192.478,275.917,-66.561,-176.917,7.249,148.464
C01463=1192.474,276.166,-66.590,-176.914,7.252,148.464
C01464=1192.470,276.414,-66.618,-176.911,7.255,148.464
C01465=1192.465,276.663,-66.646,-176.909,7.257,148.464
C01466=1192.461,276.911,-66.674,-176.906,7.260,148.464
C01467=1192.456,277.159,-66.703,-176.904,7.262,148.464
C01468=1192.453,277.407,-66.731,-176.901,7.265,148.464
C01469=1192.448,277.656,-66.760,-176.898,7.268,148.464
C01470=1192.443,277.904,-66.789,-176.896,7.270,148.464
C01471=1192.439,278.153,-66.817,-176.893,7.273,148.464
C01472=1192.435,278.401,-66.846,-176.891,7.276,148.464
C01473=1192.431,278.649,-66.874,-176.889,7.279,148.464
C01474=1192.426,278.898,-66.903,-176.885,7.281,148.463
C01475=1192.421,279.146,-66.931,-176.883,7.283,148.463
C01476=1192.418,279.394,-66.960,-176.881,7.286,148.463
C01477=1192.413,279.642,-66.988,-176.878,7.289,148.463
C01478=1192.409,279.891,-67.016,-176.876,7.292,148.463
C01479=1192.405,280.139,-67.046,-176.873,7.295,148.463
C01480=1192.400,280.387,-67.074,-176.871,7.297,148.463
C01481=1192.396,280.636,-67.102,-176.868,7.299,148.463
C01482=1192.392,280.884,-67.132,-176.865,7.302,148.463
C01483=1192.387,281.132,-67.160,-176.863,7.305,148.463
C01484=1192.383,281.380,-67.189,-176.860,7.308,148.463
C01485=1192.379,281.629,-67.218,-176.858,7.310,148.463
C01486=1192.374,281.877,-67.246,-176.855,7.313,148.463
C01487=1192.370,282.125,-67.275,-176.852,7.316,148.463
C01488=1192.366,282.374,-67.304,-176.850,7.318,148.462
C01489=1192.361,282.622,-67.333,-176.847,7.321,148.462
C01490=1192.356,282.871,-67.362,-176.844,7.324,148.462
C01491=1192.353,283.119,-67.390,-176.842,7.326,148.462
C01492=1192.348,283.367,-67.419,-176.840,7.329,148.462
C01493=1192.344,283.615,-67.448,-176.837,7.332,148.462
C01494=1192.339,283.864,-67.477,-176.835,7.334,148.462
C01495=1192.336,284.112,-67.506,-176.832,7.337,148.462
C01496=1192.331,284.360,-67.534,-176.830,7.339,148.462
C01497=1192.327,284.608,-67.564,-176.827,7.342,148.462
C01498=1192.322,284.857,-67.592,-176.824,7.345,148.462
C01499=1192.317,285.105,-67.622,-176.822,7.347,148.461
C01500=1192.314,285.354,-67.650,-176.819,7.350,148.461
C01501=1192.309,285.602,-67.679,-176.816,7.353,148.461
C01502=1192.305,285.850,-67.709,-176.814,7.355,148.461
C01503=1192.300,286.098,-67.737,-176.812,7.358,148.461
C01504=1192.296,286.347,-67.766,-176.809,7.361,148.461
C01505=1192.292,286.595,-67.796,-176.807,7.363,148.461
C01506=1192.288,286.843,-67.824,-176.804,7.366,148.461
C01507=1192.283,287.091,-67.853,-176.801,7.369,148.461
C01508=1192.279,287.339,-67.883,-176.799,7.372,148.461
C01509=1192.274,287.588,-67.911,-176.796,7.375,148.461
C01510=1192.270,287.836,-67.941,-176.794,7.378,148.461
C01511=1192.266,288.085,-67.970,-176.792,7.380,148.461
C01512=1192.261,288.359,-68.002,-176.789,7.383,148.461
C01513=1192.256,288.634,-68.034,-176.786,7.385,148.461
C01514=1192.252,288.908,-68.067,-176.783,7.388,148.461
C01515=1192.247,289.182,-68.098,-176.780,7.392,148.461
C01516=1192.243,289.431,-68.128,-176.777,7.394,148.461
C01517=1192.239,289.679,-68.157,-176.775,7.397,148.461
C01518=1192.234,289.927,-68.186,-176.772,7.400,148.461
C01519=1192.229,290.175,-68.215,-176.770,7.403,148.460
C01520=1192.225,290.424,-68.245,-176.767,7.406,148.460
C01521=1192.221,290.672,-68.274,-176.765,7.409,148.460
C01522=1192.217,290.920,-68.303,-176.762,7.411,148.460
C01523=1192.213,291.169,-68.333,-176.760,7.414,148.460
C01524=1192.209,291.417,-68.362,-176.757,7.417,148.460
C01525=1192.204,291.664,-68.391,-176.755,7.419,148.460
C01526=1192.200,291.913,-68.421,-176.752,7.422,148.460
C01527=1192.195,292.162,-68.450,-176.749,7.425,148.460
C01528=1192.191,292.410,-68.479,-176.747,7.427,148.460
C01529=1192.187,292.658,-68.509,-176.745,7.430,148.460
C01530=1192.183,292.906,-68.538,-176.742,7.433,148.460
C01531=1192.178,293.155,-68.567,-176.740,7.435,148.460
C01532=1192.174,293.403,-68.597,-176.737,7.438,148.460
C01533=1192.170,293.651,-68.626,-176.734,7.441,148.460
C01534=1192.164,293.899,-68.656,-176.732,7.444,148.460
C01535=1192.160,294.147,-68.686,-176.729,7.447,148.460
C01536=1192.156,294.396,-68.715,-176.727,7.450,148.460
C01537=1192.152,294.643,-68.745,-176.724,7.453,148.460
C01538=1192.148,294.891,-68.775,-176.722,7.455,148.460
C01539=1192.144,295.140,-68.804,-176.719,7.458,148.460
C01540=1192.140,295.388,-68.834,-176.716,7.461,148.460
C01541=1192.136,295.636,-68.863,-176.714,7.463,148.460
C01542=1192.131,295.885,-68.892,-176.712,7.466,148.460
C01543=1192.126,296.133,-68.922,-176.709,7.469,148.460
C01544=1192.122,296.381,-68.952,-176.706,7.472,148.460
C01545=1192.118,296.630,-68.981,-176.704,7.474,148.459
C01546=1192.114,296.877,-69.012,-176.701,7.477,148.459
C01547=1192.110,297.126,-69.041,-176.699,7.480,148.459
C01548=1192.105,297.374,-69.071,-176.696,7.482,148.459
C01549=1192.101,297.622,-69.100,-176.694,7.485,148.459
C01550=1192.097,297.871,-69.130,-176.691,7.488,148.459
C01551=1192.093,298.118,-69.160,-176.688,7.491,148.459
C01552=1192.089,298.367,-69.190,-176.686,7.494,148.459
C01553=1192.084,298.615,-69.220,-176.684,7.497,148.459
C01554=1192.080,298.863,-69.250,-176.681,7.500,148.459
C01555=1192.076,299.111,-69.279,-176.679,7.503,148.459
C01556=1192.071,299.359,-69.309,-176.676,7.505,148.459
C01557=1192.067,299.608,-69.339,-176.674,7.508,148.459
C01558=1192.063,299.856,-69.369,-176.671,7.511,148.459
C01559=1192.059,300.104,-69.398,-176.669,7.513,148.459
C01560=1192.054,300.352,-69.428,-176.666,7.516,148.459
C01561=1192.050,300.600,-69.459,-176.663,7.519,148.459
C01562=1192.046,300.848,-69.488,-176.661,7.522,148.459
C01563=1192.041,301.096,-69.519,-176.659,7.524,148.459
C01564=1192.037,301.345,-69.548,-176.656,7.527,148.459
C01565=1192.033,301.593,-69.578,-176.654,7.531,148.459
C01566=1192.028,301.841,-69.608,-176.651,7.534,148.459
C01567=1192.024,302.089,-69.638,-176.649,7.536,148.459
C01568=1192.020,302.337,-69.668,-176.646,7.539,148.459
C01569=1192.016,302.586,-69.699,-176.643,7.542,148.459
C01570=1192.012,302.834,-69.729,-176.641,7.545,148.459
C01571=1192.007,303.082,-69.759,-176.638,7.547,148.459
C01572=1192.003,303.330,-69.789,-176.636,7.550,148.459
C01573=1191.999,303.578,-69.818,-176.634,7.554,148.459
C01574=1191.994,303.826,-69.849,-176.631,7.557,148.459
C01575=1191.990,304.074,-69.879,-176.629,7.559,148.459
C01576=1191.985,304.322,-69.909,-176.626,7.562,148.459
C01577=1191.981,304.571,-69.939,-176.623,7.565,148.459
C01578=1191.977,304.819,-69.970,-176.621,7.568,148.459
C01579=1191.973,305.067,-69.999,-176.618,7.570,148.459
C01580=1191.969,305.315,-70.030,-176.616,7.573,148.459
C01581=1191.964,305.563,-70.060,-176.613,7.576,148.459
C01582=1191.960,305.811,-70.090,-176.611,7.579,148.459
C01583=1191.956,306.059,-70.121,-176.609,7.581,148.459
C01584=1191.952,306.307,-70.151,-176.606,7.584,148.459
C01585=1191.947,306.556,-70.181,-176.603,7.587,148.459
C01586=1191.943,306.804,-70.212,-176.601,7.591,148.459
C01587=1191.939,307.052,-70.242,-176.599,7.593,148.459
C01588=1191.934,307.300,-70.272,-176.596,7.596,148.459
C01589=1191.930,307.548,-70.302,-176.593,7.599,148.459
C01590=1191.926,307.796,-70.333,-176.591,7.602,148.459
C01591=1191.922,308.044,-70.363,-176.589,7.604,148.459
C01592=1191.917,308.293,-70.394,-176.586,7.607,148.459
C01593=1191.914,308.541,-70.424,-176.584,7.610,148.459
C01594=1191.909,308.789,-70.455,-176.581,7.614,148.459
C01595=1191.904,309.037,-70.485,-176.578,7.617,148.459
C01596=1191.900,309.285,-70.515,-176.576,7.619,148.459
C01597=1191.896,309.533,-70.546,-176.574,7.622,148.459
C01598=1191.892,309.781,-70.576,-176.571,7.625,148.459
C01599=1191.888,310.029,-70.607,-176.568,7.628,148.459
C01600=1191.883,310.277,-70.638,-176.566,7.630,148.459
C01601=1191.880,310.525,-70.668,-176.564,7.634,148.460
C01602=1191.875,310.773,-70.699,-176.561,7.637,148.460
C01603=1191.870,311.022,-70.729,-176.559,7.640,148.460
C01604=1191.866,311.270,-70.759,-176.556,7.643,148.460
C01605=1191.862,311.518,-70.790,-176.554,7.645,148.459
C01606=1191.858,311.766,-70.821,-176.552,7.648,148.460
C01607=1191.854,312.014,-70.851,-176.549,7.651,148.460
C01608=1191.849,312.262,-70.882,-176.546,7.654,148.460
C01609=1191.845,312.510,-70.913,-176.544,7.656,148.460
C01610=1191.841,312.758,-70.943,-176.542,7.660,148.460
C01611=1191.837,313.006,-70.974,-176.539,7.663,148.460
C01612=1191.833,313.255,-71.005,-176.536,7.666,148.460
C01613=1191.828,313.503,-71.036,-176.534,7.669,148.460
C01614=1191.824,313.750,-71.066,-176.532,7.671,148.460
C01615=1191.820,313.998,-71.097,-176.529,7.674,148.460
C01616=1191.815,314.275,-71.131,-176.527,7.677,148.460
C01617=1191.811,314.551,-71.166,-176.523,7.681,148.460
C01618=1191.805,314.828,-71.200,-176.521,7.684,148.460
C01619=1191.801,315.104,-71.235,-176.518,7.687,148.460
C01620=1191.797,315.352,-71.266,-176.516,7.690,148.460
C01621=1191.793,315.600,-71.296,-176.513,7.693,148.460
C01622=1191.789,315.849,-71.327,-176.511,7.696,148.460
C01623=1191.784,316.097,-71.358,-176.509,7.699,148.460
C01624=1191.780,316.344,-71.389,-176.506,7.702,148.460
C01625=1191.776,316.593,-71.420,-176.504,7.705,148.460
C01626=1191.771,316.841,-71.451,-176.501,7.708,148.460
C01627=1191.767,317.088,-71.481,-176.499,7.710,148.460
C01628=1191.763,317.337,-71.512,-176.497,7.714,148.461
C01629=1191.759,317.584,-71.544,-176.494,7.717,148.461
C01630=1191.755,317.833,-71.575,-176.491,7.720,148.461
C01631=1191.750,318.081,-71.606,-176.489,7.723,148.461
C01632=1191.746,318.329,-71.637,-176.487,7.725,148.461
C01633=1191.742,318.577,-71.668,-176.484,7.728,148.461
C01634=1191.737,318.825,-71.699,-176.482,7.732,148.461
C01635=1191.734,319.073,-71.730,-176.479,7.735,148.461
C01636=1191.730,319.321,-71.761,-176.477,7.738,148.461
C01637=1191.725,319.568,-71.792,-176.475,7.740,148.461
C01638=1191.721,319.817,-71.823,-176.472,7.743,148.461
C01639=1191.717,320.064,-71.855,-176.470,7.746,148.461
C01640=1191.713,320.313,-71.886,-176.467,7.749,148.461
C01641=1191.709,320.560,-71.917,-176.464,7.752,148.461
C01642=1191.705,320.809,-71.948,-176.463,7.755,148.461
C01643=1191.700,321.057,-71.979,-176.460,7.758,148.461
C01644=1191.696,321.305,-72.011,-176.458,7.761,148.462
C01645=1191.692,321.553,-72.042,-176.455,7.764,148.462
C01646=1191.687,321.800,-72.073,-176.452,7.767,148.462
C01647=1191.683,322.049,-72.104,-176.450,7.771,148.462
C01648=1191.679,322.296,-72.136,-176.448,7.773,148.462
C01649=1191.675,322.545,-72.167,-176.446,7.776,148.462
C01650=1191.671,322.792,-72.198,-176.443,7.779,148.462
C01651=1191.667,323.041,-72.229,-176.441,7.783,148.462
C01652=1191.662,323.288,-72.261,-176.438,7.786,148.462
C01653=1191.658,323.537,-72.292,-176.436,7.788,148.462
C01654=1191.654,323.784,-72.324,-176.434,7.791,148.462
C01655=1191.650,324.033,-72.355,-176.431,7.794,148.462
C01656=1191.646,324.280,-72.386,-176.429,7.797,148.463
C01657=1191.641,324.529,-72.419,-176.426,7.800,148.463
C01658=1191.637,324.777,-72.449,-176.424,7.804,148.463
C01659=1191.633,325.025,-72.481,-176.422,7.806,148.463
C01660=1191.629,325.273,-72.512,-176.419,7.809,148.463
C01661=1191.625,325.521,-72.544,-176.417,7.812,148.463
C01662=1191.621,325.769,-72.576,-176.414,7.816,148.463
C01663=1191.616,326.017,-72.606,-176.412,7.819,148.463
C01664=1191.613,326.265,-72.638,-176.410,7.822,148.463
C01665=1191.608,326.512,-72.670,-176.407,7.824,148.463
C01666=1191.604,326.761,-72.701,-176.405,7.827,148.464
C01667=1191.599,327.008,-72.733,-176.402,7.830,148.464
C01668=1191.596,327.256,-72.765,-176.400,7.834,148.464
C01669=1191.592,327.505,-72.797,-176.398,7.837,148.464
C01670=1191.587,327.752,-72.827,-176.396,7.839,148.464
C01671=1191.583,328.001,-72.860,-176.393,7.842,148.464
C01672=1191.578,328.248,-72.891,-176.391,7.846,148.464
C01673=1191.575,328.496,-72.923,-176.388,7.849,148.464
C01674=1191.571,328.744,-72.955,-176.386,7.852,148.464
C01675=1191.566,328.993,-72.986,-176.383,7.855,148.464
C01676=1191.562,329.241,-73.018,-176.382,7.857,148.464
C01677=1191.558,329.488,-73.050,-176.379,7.861,148.465
C01678=1191.554,329.736,-73.082,-176.377,7.864,148.465
C01679=1191.550,329.984,-73.114,-176.374,7.867,148.465
C01680=1191.545,330.232,-73.145,-176.372,7.870,148.465
C01681=1191.542,330.480,-73.177,-176.369,7.873,148.465
C01682=1191.536,330.727,-73.209,-176.368,7.876,148.465
C01683=1191.532,330.976,-73.241,-176.365,7.879,148.465
C01684=1191.529,331.224,-73.272,-176.363,7.882,148.466
C01685=1191.524,331.471,-73.304,-176.360,7.885,148.466
C01686=1191.520,331.720,-73.336,-176.358,7.889,148.466
C01687=1191.516,331.968,-73.368,-176.356,7.892,148.466
C01688=1191.512,332.215,-73.400,-176.354,7.894,148.466
C01689=1191.508,332.463,-73.432,-176.351,7.897,148.466
C01690=1191.504,332.711,-73.464,-176.349,7.900,148.466
C01691=1191.499,332.959,-73.496,-176.346,7.904,148.466
C01692=1191.495,333.207,-73.528,-176.344,7.907,148.467
C01693=1191.491,333.455,-73.560,-176.341,7.910,148.467
C01694=1191.487,333.704,-73.592,-176.339,7.913,148.467
C01695=1191.483,333.950,-73.624,-176.337,7.916,148.467
C01696=1191.479,334.199,-73.657,-176.335,7.919,148.467
C01697=1191.475,334.447,-73.689,-176.333,7.922,148.467
C01698=1191.470,334.694,-73.720,-176.330,7.926,148.467
C01699=1191.466,334.942,-73.753,-176.328,7.929,148.467
C01700=1191.462,335.190,-73.784,-176.325,7.932,148.468
C01701=1191.458,335.439,-73.817,-176.324,7.934,148.468
C01702=1191.454,335.686,-73.848,-176.321,7.938,148.468
C01703=1191.449,335.934,-73.881,-176.319,7.941,148.468
C01704=1191.446,336.182,-73.913,-176.316,7.944,148.468
C01705=1191.441,336.430,-73.946,-176.314,7.947,148.468
C01706=1191.437,336.678,-73.977,-176.312,7.951,148.469
C01707=1191.433,336.926,-74.010,-176.310,7.953,148.469
C01708=1191.429,337.173,-74.042,-176.308,7.956,148.469
C01709=1191.425,337.422,-74.075,-176.305,7.960,148.469
C01710=1191.420,337.669,-74.106,-176.303,7.963,148.469
C01711=1191.416,337.917,-74.139,-176.300,7.966,148.469
C01712=1191.413,338.165,-74.171,-176.298,7.969,148.469
C01713=1191.408,338.413,-74.204,-176.296,7.973,148.470
C01714=1191.404,338.660,-74.235,-176.294,7.975,148.470
C01715=1191.400,338.908,-74.268,-176.292,7.978,148.470
C01716=1191.396,339.156,-74.300,-176.289,7.981,148.470
C01717=1191.392,339.405,-74.332,-176.287,7.985,148.470
C01718=1191.387,339.652,-74.366,-176.285,7.988,148.470
C01719=1191.384,339.900,-74.397,-176.283,7.991,148.471
C01720=1191.379,340.178,-74.434,-176.280,7.995,148.471
C01721=1191.374,340.457,-74.470,-176.278,7.998,148.471
C01722=1191.370,340.735,-74.507,-176.275,8.002,148.471
C01723=1191.364,341.015,-74.543,-176.273,8.005,148.471
C01724=1191.361,341.262,-74.576,-176.270,8.009,148.472
C01725=1191.356,341.511,-74.608,-176.268,8.012,148.472
C01726=1191.352,341.758,-74.641,-176.266,8.015,148.472
C01727=1191.349,342.006,-74.673,-176.264,8.018,148.472
C01728=1191.344,342.253,-74.706,-176.262,8.021,148.472
C01729=1191.339,342.502,-74.739,-176.259,8.024,148.472
C01730=1191.336,342.749,-74.771,-176.257,8.027,148.473
C01731=1191.331,342.997,-74.804,-176.255,8.031,148.473
C01732=1191.327,343.245,-74.837,-176.253,8.034,148.473
C01733=1191.324,343.493,-74.869,-176.251,8.037,148.473
C01734=1191.319,343.741,-74.902,-176.249,8.040,148.474
C01735=1191.315,343.989,-74.934,-176.246,8.043,148.474
C01736=1191.310,344.236,-74.967,-176.244,8.047,148.474
C01737=1191.307,344.484,-74.999,-176.242,8.050,148.474
C01738=1191.302,344.732,-75.032,-176.240,8.053,148.474
C01739=1191.298,344.980,-75.065,-176.237,8.057,148.475
C01740=1191.294,345.228,-75.098,-176.236,8.059,148.475
C01741=1191.290,345.476,-75.131,-176.233,8.062,148.475
C01742=1191.286,345.723,-75.163,-176.231,8.066,148.475
C01743=1191.282,345.971,-75.196,-176.229,8.069,148.475
C01744=1191.278,346.219,-75.229,-176.227,8.072,148.476
C01745=1191.274,346.467,-75.262,-176.225,8.076,148.476
C01746=1191.269,346.715,-75.295,-176.222,8.079,148.476
C01747=1191.266,346.963,-75.327,-176.221,8.081,148.476
C01748=1191.261,347.210,-75.360,-176.218,8.085,148.476
C01749=1191.257,347.458,-75.393,-176.216,8.088,148.477
C01750=1191.253,347.705,-75.426,-176.214,8.091,148.477
C01751=1191.249,347.953,-75.459,-176.212,8.095,148.477
C01752=1191.244,348.201,-75.492,-176.209,8.098,148.477
C01753=1191.241,348.449,-75.524,-176.207,8.101,148.478
C01754=1191.237,348.697,-75.557,-176.205,8.104,148.478
C01755=1191.233,348.944,-75.591,-176.203,8.107,148.478
C01756=1191.228,349.192,-75.624,-176.201,8.111,148.478
C01757=1191.224,349.440,-75.656,-176.199,8.114,148.479
C01758=1191.220,349.688,-75.689,-176.197,8.118,148.479
C01759=1191.216,349.936,-75.722,-176.195,8.121,148.479
C01760=1191.212,350.184,-75.756,-176.192,8.124,148.479
C01761=1191.207,350.431,-75.789,-176.191,8.127,148.479
C01762=1191.203,350.679,-75.822,-176.189,8.130,148.480
C01763=1191.199,350.927,-75.855,-176.187,8.134,148.480
C01764=1191.195,351.175,-75.888,-176.184,8.137,148.480
C01765=1191.191,351.422,-75.921,-176.182,8.140,148.481
C01766=1191.187,351.670,-75.954,-176.180,8.144,148.481
C01767=1191.183,351.917,-75.987,-176.178,8.147,148.481
C01768=1191.179,352.165,-76.020,-176.177,8.150,148.481
C01769=1191.175,352.413,-76.053,-176.174,8.153,148.482
C01770=1191.171,352.661,-76.087,-176.172,8.156,148.482
C01771=1191.167,352.909,-76.120,-176.170,8.160,148.482
C01772=1191.163,353.157,-76.153,-176.168,8.163,148.483
C01773=1191.159,353.404,-76.186,-176.166,8.167,148.483
C01774=1191.155,353.652,-76.220,-176.164,8.169,148.483
C01775=1191.150,353.900,-76.253,-176.162,8.172,148.483
C01776=1191.146,354.148,-76.286,-176.160,8.176,148.484
C01777=1191.142,354.396,-76.320,-176.158,8.179,148.484
C01778=1191.138,354.643,-76.353,-176.156,8.183,148.484
C01779=1191.133,354.891,-76.386,-176.154,8.186,148.484
C01780=1191.130,355.138,-76.420,-176.152,8.190,148.485
C01781=1191.126,355.386,-76.453,-176.150,8.192,148.485
C01782=1191.122,355.634,-76.486,-176.148,8.196,148.485
C01783=1191.118,355.882,-76.520,-176.146,8.199,148.486
C01784=1191.114,356.130,-76.553,-176.144,8.203,148.486
C01785=1191.110,356.377,-76.587,-176.142,8.206,148.486
C01786=1191.106,356.625,-76.620,-176.140,8.209,148.486
C01787=1191.101,356.873,-76.654,-176.138,8.213,148.487
C01788=1191.097,357.120,-76.687,-176.136,8.216,148.487
C01789=1191.093,357.368,-76.720,-176.134,8.219,148.487
C01790=1191.089,357.616,-76.754,-176.132,8.223,148.488
C01791=1191.085,357.864,-76.787,-176.130,8.226,148.488
C01792=1191.081,358.111,-76.820,-176.128,8.230,148.488
C01793=1191.077,358.359,-76.854,-176.126,8.233,148.489
C01794=1191.072,358.607,-76.888,-176.124,8.236,148.489
C01795=1191.068,358.854,-76.921,-176.122,8.239,148.489
C01796=1191.065,359.102,-76.955,-176.120,8.243,148.490
C01797=1191.061,359.350,-76.989,-176.118,8.246,148.490
C01798=1191.057,359.598,-77.022,-176.116,8.250,148.490
C01799=1191.052,359.845,-77.056,-176.114,8.253,148.490
C01800=1191.048,360.093,-77.089,-176.113,8.256,148.491
C01801=1191.044,360.341,-77.123,-176.111,8.259,148.491
C01802=1191.041,360.588,-77.157,-176.109,8.263,148.492
C01803=1191.037,360.836,-77.190,-176.107,8.266,148.492
C01804=1191.032,361.083,-77.224,-176.105,8.270,148.492
C01805=1191.028,361.331,-77.258,-176.104,8.272,148.493
C01806=1191.025,361.579,-77.292,-176.102,8.276,148.493
C01807=1191.020,361.827,-77.326,-176.100,8.279,148.493
C01808=1191.016,362.074,-77.359,-176.098,8.283,148.494
C01809=1191.012,362.322,-77.393,-176.096,8.287,148.494
C01810=1191.008,362.570,-77.427,-176.095,8.289,148.494
C01811=1191.004,362.818,-77.461,-176.093,8.293,148.495
C01812=1191.000,363.065,-77.494,-176.091,8.296,148.495
C01813=1190.996,363.313,-77.528,-176.089,8.300,148.496
C01814=1190.992,363.561,-77.562,-176.087,8.302,148.496
C01815=1190.988,363.808,-77.596,-176.085,8.306,148.496
C01816=1190.984,364.056,-77.629,-176.084,8.310,148.497
C01817=1190.979,364.304,-77.663,-176.082,8.313,148.497
C01818=1190.976,364.551,-77.697,-176.081,8.316,148.497
C01819=1190.972,364.798,-77.731,-176.078,8.319,148.498
C01820=1190.967,365.047,-77.765,-176.077,8.323,148.498
C01821=1190.964,365.294,-77.799,-176.075,8.326,148.498
C01822=1190.960,365.542,-77.832,-176.074,8.330,148.499
C01823=1190.955,365.789,-77.867,-176.072,8.333,148.499
